Omron CX-Programmer project NewProject (CX-Programmer 9.75)

# PLC NewPLC1: CP2E-N N

## Global symbols (name address type ; comment)
ABNRML_INDICATOR 101.06 BOOL  ; ABNORMAL_IND
AIR_PRESS_OK 0.01 BOOL  ; AIR_PRESS_OK
AUTO_SS 1.09 BOOL  ; AUTO SS
1.08 BOOL  ; manual_press
4 CHANNEL  ; LVDT1_INP_POS
5 CHANNEL  ; LVDT2_INP_POS
D100 CHANNEL  ; LVDT1_CURRENT_VAL_MM
D1000 CHANNEL  ; lvdt1_max_hmi_log
D1002 CHANNEL  ; lvdt1_min_hmi_log
D1004 CHANNEL  ; lvdt2_max_hmi_log
D1006 CHANNEL  ; lvdt2_min_hmi_log
D1010 CHANNEL  ; lvdt1_max_hmi_log.
D1012 CHANNEL  ; lvdt1_min_hmi_log.
D1014 CHANNEL  ; lvdt2_max_hmi_log.
D1016 CHANNEL  ; lvdt2_min_hmi_log.
D110 CHANNEL  ; LVDT2_CURRENT_VAL_MM
D1230 CHANNEL  ; servo_pulse.
D1240 CHANNEL  ; LVDT1_CURRENT_VAL_MM.
D1250 CHANNEL  ; LVDT2_CURRENT_VAL_MM.
D1280 CHANNEL  ; LVDT_POS_OK_PART
D1300 CHANNEL  ; rpm_hmi
D1305 CHANNEL  ; .
D1310 CHANNEL  ; servo_freq.
D150 CHANNEL  ; TOTAL PULSES FOR ROTATION
D1520 CHANNEL  ; PART2_CAL
D1550 CHANNEL  ; PART2_CAL.
D1700 CHANNEL  ; SERVO_PV
D20 CHANNEL  ; CYCLE TIME
D200 CHANNEL  ; UPPER_LIMIT_M1_HMI
D2000 CHANNEL  ; TOTAL_NG_GEAR_RUNOUT_LOWER_LIM
D2002 CHANNEL  ; TOTAL_NG_GEAR_RUNOUT_UPPER_LIM
D202 CHANNEL  ; LOWER_LIMIT_1_HMI
D204 CHANNEL  ; UPPER_LIMIT_M2_HMI
D206 CHANNEL  ; LOWER_LIMIT_M2_HMI
D210 CHANNEL  ; OFFSET_M1_HMI
D212 CHANNEL  ; OFFSET._M1_HMI
D214 CHANNEL  ; OFFSET_M2_HMI
D216 CHANNEL  ; OFFSET._M2_HMI
D22 CHANNEL  ; OK_COUNT
D220 CHANNEL  ; FINAL_UPPER_LIMIT
D222 CHANNEL  ; FINAL_LOWER_LIMIT
D224 CHANNEL  ; FINAL_LOWER_LIMIT
D230 CHANNEL  ; LOWER_LIMIT_1_HMI
D240 CHANNEL  ; LOWER_LIMIT_1_HMI
D25 CHANNEL  ; NG_COUNT
D250 CHANNEL  ; UPPER_LIMIT_M2_HMI
D260 CHANNEL  ; OFFSET_M2_HMI
D270 CHANNEL  ; LOWER_LIMIT_M2_HMI
D280 CHANNEL  ; OFFSET._M2_HMI
D300 CHANNEL  ; WORD LAMP STATUS
D550 CHANNEL  ; LVDT1_INP_POS.
D555 CHANNEL  ; LVDT2_INP_POS.
D570 CHANNEL  ; OFFSET_LVDT
D575 CHANNEL  ; LVDT2_CUR_VAL
D590 CHANNEL  ; OFFSET
D595 CHANNEL  ; LVDT1_CUR_VAL
D605 CHANNEL  ; .
D7055 CHANNEL  ; LVDT1_MAX_HMI
D820 CHANNEL  ; rot_degree
D830 CHANNEL  ; PART1_SERVOCOUNT_HMI
D840 CHANNEL  ; PART2_SERVOCOUNT_HMI
D850 CHANNEL  ; rot_deg.
D900 CHANNEL  ; LVDT2_MAX_HMI
D902 CHANNEL  ; LVDT1_MAX_HMI
D904 CHANNEL  ; LVDT2_MIN_HMI
D906 CHANNEL  ; LVDT1_Min_HMI
D910 CHANNEL  ; LVDT2_MAX_HMI
D910 CHANNEL  ; LVDT1_MAX_HMI
D920 CHANNEL  ; servo_float
D930 CHANNEL  ; part1_fullbody_servocount
D930 CHANNEL  ; PART1_FULLBODY_PULSE
D940 CHANNEL  ; PART2_FULLBODY_SERVOCOUNT
D950 CHANNEL  ; LVDT1_Min_HMI
T046 BOOL  ; delay time for lvdt to adjust
W10.00 BOOL  ; CYCLE START
W11.00 BOOL  ; PART_FEEDER_UP_BIT
W11.01 BOOL  ; PART_HOLDER_FWD_BIT
W11.02 BOOL  ; PART_FEED_DONE_FLAG
W11.03 BOOL  ; TEST_CYCLE_START
W11.04 BOOL  ; LVDT_TEST_POSITION
W11.05 BOOL  ; SERVO_CMD1
W11.06 BOOL  ; TEST_DONE_FLAG_OK
W11.07 BOOL  ; CYCLE_COMPLETING_OK_process_start
W11.08 BOOL  ; PART_FEEDER_UP_OK
W11.09 BOOL  ; CYCLE_COM_OK_flag
W11.10 BOOL  ; LVDT_PUSHER_FWD_OK
W12.00 BOOL  ; TYPENO._1
W12.01 BOOL  ; TYPNO._2
W12.02 BOOL  ; PART1
W12.03 BOOL  ; PART2
W13.06 BOOL  ; TEST_DONE_FLAG_NG
W13.07 BOOL  ; CYCLE_COMPLETING_NG_process_start
W13.08 BOOL  ; PART_FEEDER_UP_NG
W13.09 BOOL  ; CYCLE_COM_NG
W13.10 BOOL  ; LVDT_PUSHER_fwd_NG
W14.00 BOOL  ; BIO_SCAN_OK
W15.00 BOOL  ; NG_FLAG
W15.01 BOOL  ; OK_FLAG
W16.00 BOOL  ; PART_FEEDER_DN_BIT
W16.01 BOOL  ; PART_HOLDER_REV_BIT
W16.04 BOOL  ; LVDT_CYL_REV_ok
W16.08 BOOL  ; PART_FEED_DN_BIT_OK
W16.10 BOOL  ; LVDT_PUSHER_REV_BIT
W17.01 BOOL  ; PART_HOLDER_REV__NG_BIT
W17.04 BOOL  ; LVDT_CYL_REV_NG
W17.08 BOOL  ; PART_FEEDER_DN_NG
W17.10 BOOL  ; LVDT_PUSHER_REV_NG
W18.04 BOOL  ; LVDT_CYL_REV_EMG
W19.00 BOOL  ; BUZZER_NG_PART
W19.01 BOOL  ; BUZZER_BIT
W19.03 BOOL  ; ng_bin_sensor
W22.00 BOOL  ; PART_FEED_UP_MAN
W22.01 BOOL  ; PART_FEED_DN_MAN
W22.02 BOOL  ; PART_HOLD1_FWD_MAN
W22.03 BOOL  ; PART_HOLD2_FWD_MAN
W22.04 BOOL  ; PART_HOLD1_REV_MAN
W22.05 BOOL  ; PART_HOLD2_REV_MAN
W22.06 BOOL  ; LVDT_FWD_MAN
W22.07 BOOL  ; LVDT_REV_MAN
W22.08 BOOL  ; LVDT_PUSH_FWD_MAN
W22.09 BOOL  ; LVDT_PUSH_REV_MAN
W23.00 BOOL  ; PART_FEED_UP_MAN
W23.01 BOOL  ; PART_FEED_DN_MAN
W23.02 BOOL  ; PART_HOLD1_FWD_MAN
W23.03 BOOL  ; PART_HOLD2_FWD_MAN
W23.04 BOOL  ; PART_HOLD1_REV_MAN
W23.05 BOOL  ; PART_HOLD2_REV_MAN
W23.06 BOOL  ; LVDT_FWD_MAN
W23.07 BOOL  ; LVDT_REV_MAN
W23.08 BOOL  ; LVDT_PUSH_FWD_MAN
W23.09 BOOL  ; LVDT_PUSH_REV_MAN
W24.00 BOOL  ; FULL_PART_TESTED
W25.00 BOOL  ; LVDT_ORIGIN
W25.01 BOOL  ; PART_HOLDER_ORIGIN
W25.02 BOOL  ; PART_FEEDER_ORIGIN
W25.03 BOOL  ; LVDT_PUSHER_FWD
W25.04 BOOL  ; LVDT_PUSHER_HM
W25.12 BOOL  ; part_feeder_up_org
W25.15 BOOL  ; PUSHER_HOME_ORG
W26.00 BOOL  ; MASTER_ON_BIT
W26.01 BOOL  ; SERVO_MAN
W26.02 BOOL  ; LVDT_HOME
W26.12 BOOL  ; servo_man
W2.06 BOOL  ; BIO_SCANNED
W2.08 BOOL  ; RESET_ORG
W30.00 BOOL  ; COUNTER_RESET_HMI
W32.00 BOOL  ; servo_cmd2
W39.01 BOOL  ; WRONG MODEL SELECTED
W50.00 BOOL  ; PART_FEEDER_UP_RS_ABS/ CYL NOT UP
W50.01 BOOL  ; PART_FEEDER_DN_RS_ABS/CYL NOT DN
W50.02 BOOL  ; PART_HOLD_CLOSE_RS_ABS/ PART NOT HOLD
W50.03 BOOL  ; PART_HOLD_OPEN_RS_ABS/ PART NOT RELEASED
W50.04 BOOL  ; LVDT1_TEST_RS_ABS/ LVDT1 NOT AT TEST POS
W50.05 BOOL  ; LVDT2_TEST_RS_ABS/ LVDT2 NOT AT TEST POS
W50.06 BOOL  ; LVDT1_HM_RS_ABS/ LVDT1 NOT AT HOME POS
W50.07 BOOL  ; LVDT2_HM_RS_ABS/ LVDT2 NOT AT HOME POS
W50.08 BOOL  ; PUSHER LIM RS ABS / PUSHER NOT MOVING FWD
W50.09 BOOL  ; PUSHER HOME RS ABSENT / PUSHER NOT MOVING REV
W50.10 BOOL  ; CHECK_PART_CLAMP_RS/PART SELECTION RS ERROR
W55.00 BOOL  ; servo_run1_complete_flag
W55.01 BOOL  ; lvdt_ready_for_test
W55.02 BOOL  ; NGpart_ready_to_remove
W55.03 BOOL  ; OKpart_ready_to_remove
W55.04 BOOL  ; LVDT_PUSHING_DONE
W55.05 BOOL  ; PAR_UNCLAMP_DONE_OK
W55.06 BOOL  ; LVDT_PUSH_DONE_NG
W55.07 BOOL  ; PAR_UNCLAMP_DONE_NG
W55.08 BOOL  ; NGpart_ready_to_remove
W55.10 BOOL  ; lvdt_home
W56.01 BOOL  ; servo_ready_for_cmd2
W60.10 BOOL  ; PART_NOT_MATCHED
W60.11 BOOL  ; PART1_MATCHED
W60.12 BOOL  ; PART_2_MATCHED
W6.00 BOOL  ; LOG_PART1_RESULT
W6.01 BOOL  ; LOG_PART2_RESULT
W70.00 BOOL  ; EMG_ALARM
W70.01 BOOL  ; AIR_PRESS_ALARM
W70.02 BOOL  ; SAFETY_DOOR_ALARM
W70.03 BOOL  ; PART_ABSENT_ALARM
W70.04 BOOL  ; PART_NOT_MATCH_ALARM
W76.01 BOOL  ; part2_match
W77.01 BOOL  ; not_match
W78.01 BOOL  ; not_match.
W79.01 BOOL  ; part1_match
W80.00 BOOL  ; ABNORMAL_LIGHT
W80.03 BOOL  ; PART_NOT_PRESENT_ALARM
W80.04 BOOL  ; NG_PART_ALARM
W8.00 BOOL  ; LVDT_PUSHED_flag
W8.01 BOOL  ; LVDT_PUSH_DONE
W9.00 BOOL  ; MACHINE_HOME
W9.01 BOOL  ; LVDT_PUSH_ONCE
W9.02 BOOL  ; LVDT_PUSH_RTN
W9.03 BOOL  ; LVDT_PUSHED_FLAG
W9.04 BOOL  ; CYCLE READY_FLAG
W9.05 BOOL  ; servo_cmd3
W9.06 BOOL  ; part_ok_HMI
W9.07 BOOL  ; part_ng_HMI
BIO_SCAN 0.00 BOOL  ; BIOMETRIC
DUAL_PB1 1.11 BOOL  ; DUAL_PB1
DUAL_PB2 2.00 BOOL  ; DUAL_PB2
EMG_LAMP 101.03 BOOL  ; EMG_LAMP
EMG_PB 2.04 BOOL  ; EMG_PB
LVDT1_HOME_RS 0.05 BOOL  ; LVDT1_HM_RS
LVDT1_TEST_RS 0.04 BOOL  ; LVDT1_TST_RS
LVDT2_HOME_RS 0.07 BOOL  ; LVDT2_HM_RS
LVDT2_TEST_RS 0.06 BOOL  ; LVDT2_TST_RS
LVDT_CYL_FWD 100.06 BOOL  ; LVDT_CYL_FWD
LVDT_CYL_REV 100.07 BOOL  ; LVDT_CYL_REV
LVDT_PUSHER_FWD 101.00 BOOL  ; LVDT_PUSH_CYL_FWD
LVDT_PUSHER_REV 101.01 BOOL  ; LVDT_PUSH_CYL_REV
LVDT_PUSH_HOME 2.06 BOOL  ; LVDT_PUSH_HOME
LVDT_PUSH_LIM 2.05 BOOL  ; LVDT_PUSHER_LIM
MANUAL_SS 1.10 BOOL  ; MANUAL_SS
MASTER_LAMP 101.04 BOOL  ; MASTER_LAMP
MODEL_2 1.02 BOOL  ; 2
NG_BIN_SEN 0.11 BOOL  ; NG_BIN_SENSOR
NG_BUZZER 101.02 BOOL  ; NG_BUZZER
NG_UNCLAMP_PB 2.02 BOOL  ; NG_UNCLAMP_PB
ORGN_INDICATOR 101.05 BOOL  ; ORIGIN_IND
ORIGIN_RETURN_PB 2.01 BOOL  ; ORIGIN_RETURN_PB
PART_1 1.00 BOOL  ; PART_1
PART_2 1.01 BOOL  ; PART_2
PART_CLAMP_CLOSE_P2 2.10 BOOL  ; PART_CLAMP_CLOSE_P2
PART_FEEDER_DN 103.01 BOOL  ; PART_FEEDER_DOWN
PART_FEEDER_UP 103.00 BOOL  ; PART_FEEDER_UP
PART_FEED_DN_RS 2.08 BOOL  ; PART_FEEDER_DN_RS
PART_FEED_UP_RS 2.07 BOOL  ; PART_FEEDER_UP_RS
PART_HOLD1_CLOSE_RS 0.02 BOOL  ; PART_HOLDER_FRONT_RS
PART_HOLD1_OPEN_RS 0.03 BOOL  ; PART_HOLDER_BACK_RS
PART_HOLD2_CLOSE_RS 0.08 BOOL  ; part_holde2_close_rs
PART_HOLD2_OPEN_RS 0.09 BOOL  ; part_holder2_open_rs
PART_HOLDER1_FWD 100.01 BOOL  ; PART_HOLDER1_FWD
PART_HOLDER1_REV 100.03 BOOL  ; PART_HOLDER1_REV
PART_HOLDER2_FWD 100.04 BOOL  ; PART_HOLDER2_FWD
PART_HOLDER2_REV 100.05 BOOL  ; PART_HOLDER2_REV
PART_PRESENCE_SENSOR 2.11 BOOL  ; PART_PRESENCE_SENSOR
RESET_PB 2.03 BOOL  ; RESET_PB
SAFETY_LIM1 2.09 BOOL  ; SAFETY_LIM1
SERVO_DIR 100.01 BOOL  ; SERVO_DIRECTION
SERVO_OUT 102.04 BOOL  ; SERVO
SERVO_PULSE 100.00 BOOL  ; SERVO_PULSE
TEST_READY_SENSOR 3.00 BOOL  ; PART_READY FOR TEST SENSOR
TOWER_LIGHT 101.07 BOOL  ; TOWER_LIGHT
master_start 0.10 BOOL  ; START_PB

## Program NewProgram1 (cyclic task 0)
Local symbols
ILC BOOL
MODEL_3 BOOL
PART_UNHOLD BOOL
cf11e BOOL
dsc BOOL

### Section IN_OUT

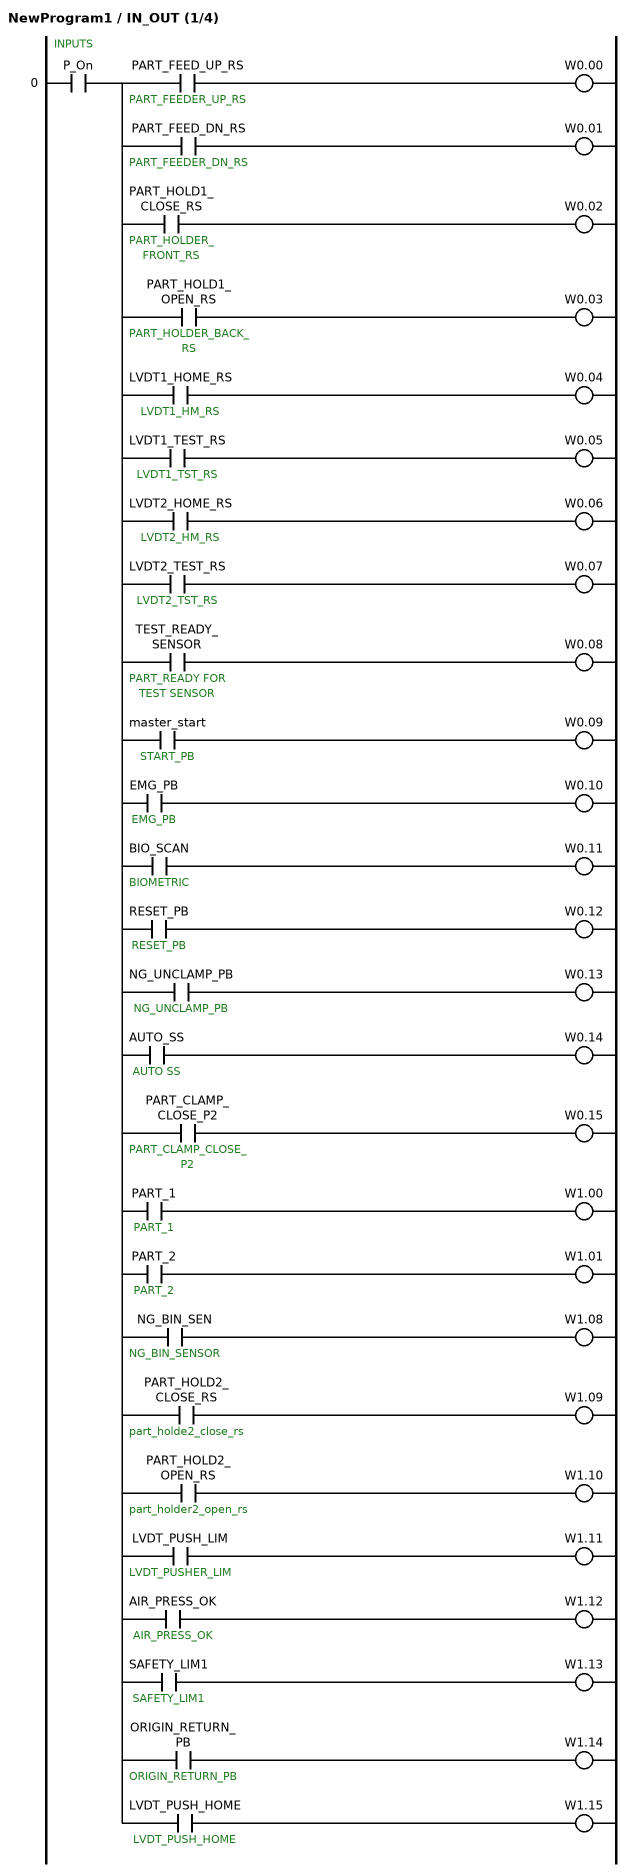
; rung 0: INPUTS
LD P_On
OUT TR0
AND PART_FEED_UP_RS  ; PART_FEEDER_UP_RS
OUT W0.00
LD TR0
AND PART_FEED_DN_RS  ; PART_FEEDER_DN_RS
OUT W0.01
LD TR0
AND PART_HOLD1_CLOSE_RS  ; PART_HOLDER_FRONT_RS
OUT W0.02
LD TR0
AND PART_HOLD1_OPEN_RS  ; PART_HOLDER_BACK_RS
OUT W0.03
LD TR0
AND LVDT1_HOME_RS  ; LVDT1_HM_RS
OUT W0.04
LD TR0
AND LVDT1_TEST_RS  ; LVDT1_TST_RS
OUT W0.05
LD TR0
AND LVDT2_HOME_RS  ; LVDT2_HM_RS
OUT W0.06
LD TR0
AND LVDT2_TEST_RS  ; LVDT2_TST_RS
OUT W0.07
LD TR0
AND TEST_READY_SENSOR  ; PART_READY FOR TEST SENSOR
OUT W0.08
LD TR0
AND master_start  ; START_PB
OUT W0.09
LD TR0
AND EMG_PB  ; EMG_PB
OUT W0.10
LD TR0
AND BIO_SCAN  ; BIOMETRIC
OUT W0.11
LD TR0
AND RESET_PB  ; RESET_PB
OUT W0.12
LD TR0
AND NG_UNCLAMP_PB  ; NG_UNCLAMP_PB
OUT W0.13
LD TR0
AND AUTO_SS  ; AUTO SS
OUT W0.14
LD TR0
AND PART_CLAMP_CLOSE_P2  ; PART_CLAMP_CLOSE_P2
OUT W0.15
LD TR0
AND PART_1  ; PART_1
OUT W1.00
LD TR0
AND PART_2  ; PART_2
OUT W1.01
LD TR0
AND NG_BIN_SEN  ; NG_BIN_SENSOR
OUT W1.08
LD TR0
AND PART_HOLD2_CLOSE_RS  ; part_holde2_close_rs
OUT W1.09
LD TR0
AND PART_HOLD2_OPEN_RS  ; part_holder2_open_rs
OUT W1.10
LD TR0
AND LVDT_PUSH_LIM  ; LVDT_PUSHER_LIM
OUT W1.11
LD TR0
AND AIR_PRESS_OK  ; AIR_PRESS_OK
OUT W1.12
LD TR0
AND SAFETY_LIM1  ; SAFETY_LIM1
OUT W1.13
LD TR0
AND ORIGIN_RETURN_PB  ; ORIGIN_RETURN_PB
OUT W1.14
LD TR0
AND LVDT_PUSH_HOME  ; LVDT_PUSH_HOME
OUT W1.15

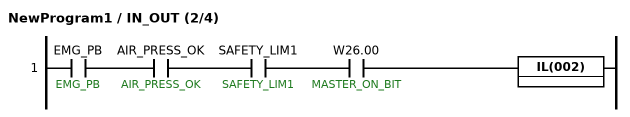
; rung 1
LD EMG_PB  ; EMG_PB
AND AIR_PRESS_OK  ; AIR_PRESS_OK
AND SAFETY_LIM1  ; SAFETY_LIM1
AND W26.00  ; MASTER_ON_BIT
IL(002)

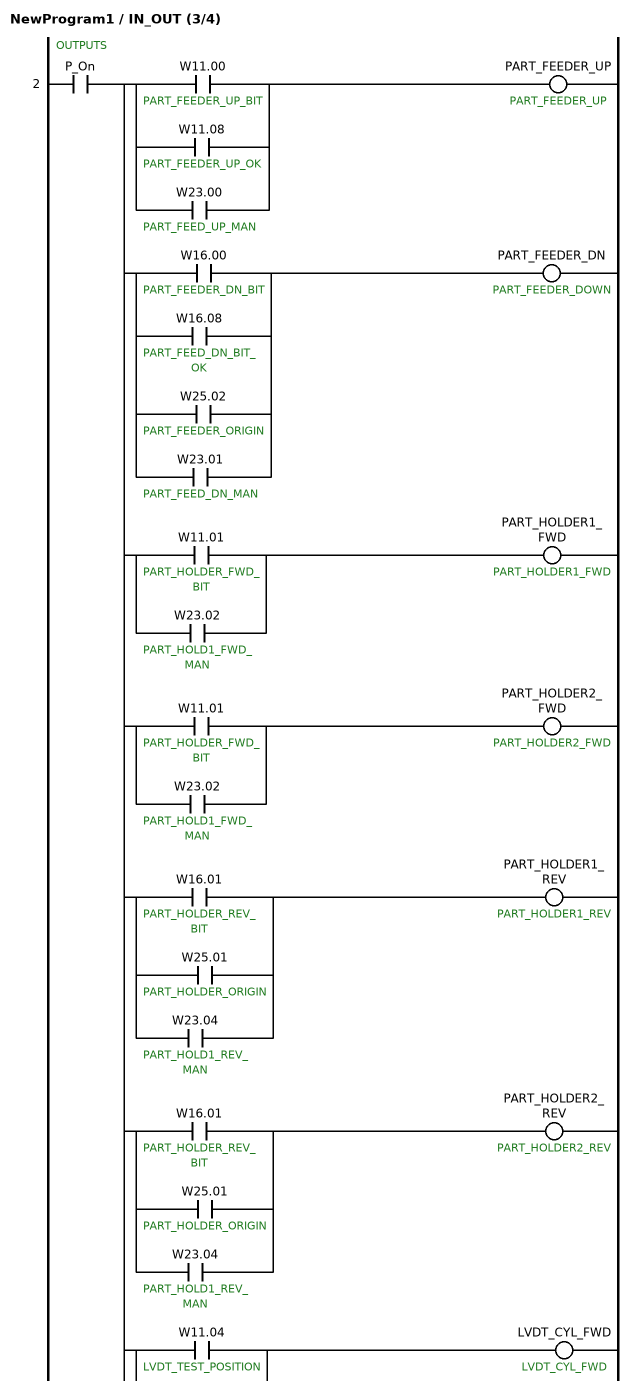

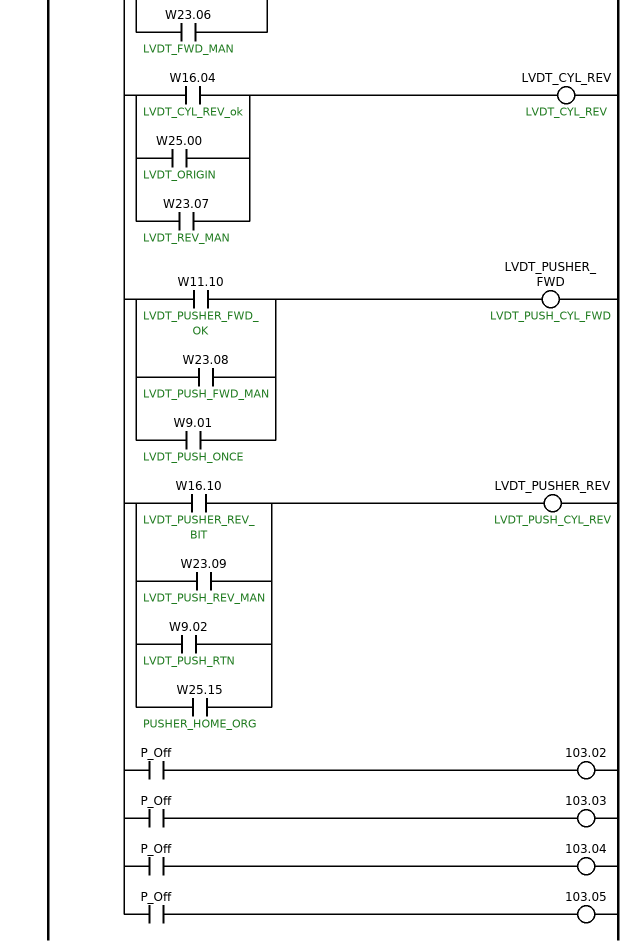
; rung 2: OUTPUTS
LD P_On
OUT TR0
LD W11.00  ; PART_FEEDER_UP_BIT
OR W11.08  ; PART_FEEDER_UP_OK
OR W23.00  ; PART_FEED_UP_MAN
ANDLD
OUT PART_FEEDER_UP  ; PART_FEEDER_UP
LD TR0
LD W16.00  ; PART_FEEDER_DN_BIT
OR W16.08  ; PART_FEED_DN_BIT_OK
OR W25.02  ; PART_FEEDER_ORIGIN
OR W23.01  ; PART_FEED_DN_MAN
ANDLD
OUT PART_FEEDER_DN  ; PART_FEEDER_DOWN
LD TR0
LD W11.01  ; PART_HOLDER_FWD_BIT
OR W23.02  ; PART_HOLD1_FWD_MAN
ANDLD
OUT PART_HOLDER1_FWD  ; PART_HOLDER1_FWD
LD TR0
LD W11.01  ; PART_HOLDER_FWD_BIT
OR W23.02  ; PART_HOLD1_FWD_MAN
ANDLD
OUT PART_HOLDER2_FWD  ; PART_HOLDER2_FWD
LD TR0
LD W16.01  ; PART_HOLDER_REV_BIT
OR W25.01  ; PART_HOLDER_ORIGIN
OR W23.04  ; PART_HOLD1_REV_MAN
ANDLD
OUT PART_HOLDER1_REV  ; PART_HOLDER1_REV
LD TR0
LD W16.01  ; PART_HOLDER_REV_BIT
OR W25.01  ; PART_HOLDER_ORIGIN
OR W23.04  ; PART_HOLD1_REV_MAN
ANDLD
OUT PART_HOLDER2_REV  ; PART_HOLDER2_REV
LD TR0
LD W11.04  ; LVDT_TEST_POSITION
OR W23.06  ; LVDT_FWD_MAN
ANDLD
OUT LVDT_CYL_FWD  ; LVDT_CYL_FWD
LD TR0
LD W16.04  ; LVDT_CYL_REV_ok
OR W25.00  ; LVDT_ORIGIN
OR W23.07  ; LVDT_REV_MAN
ANDLD
OUT LVDT_CYL_REV  ; LVDT_CYL_REV
LD TR0
LD W11.10  ; LVDT_PUSHER_FWD_OK
OR W23.08  ; LVDT_PUSH_FWD_MAN
OR W9.01  ; LVDT_PUSH_ONCE
ANDLD
OUT LVDT_PUSHER_FWD  ; LVDT_PUSH_CYL_FWD
LD TR0
LD W16.10  ; LVDT_PUSHER_REV_BIT
OR W23.09  ; LVDT_PUSH_REV_MAN
OR W9.02  ; LVDT_PUSH_RTN
OR W25.15  ; PUSHER_HOME_ORG
ANDLD
OUT LVDT_PUSHER_REV  ; LVDT_PUSH_CYL_REV
LD TR0
AND P_Off
OUT 103.02
LD TR0
AND P_Off
OUT 103.03
LD TR0
AND P_Off
OUT 103.04
LD TR0
AND P_Off
OUT 103.05

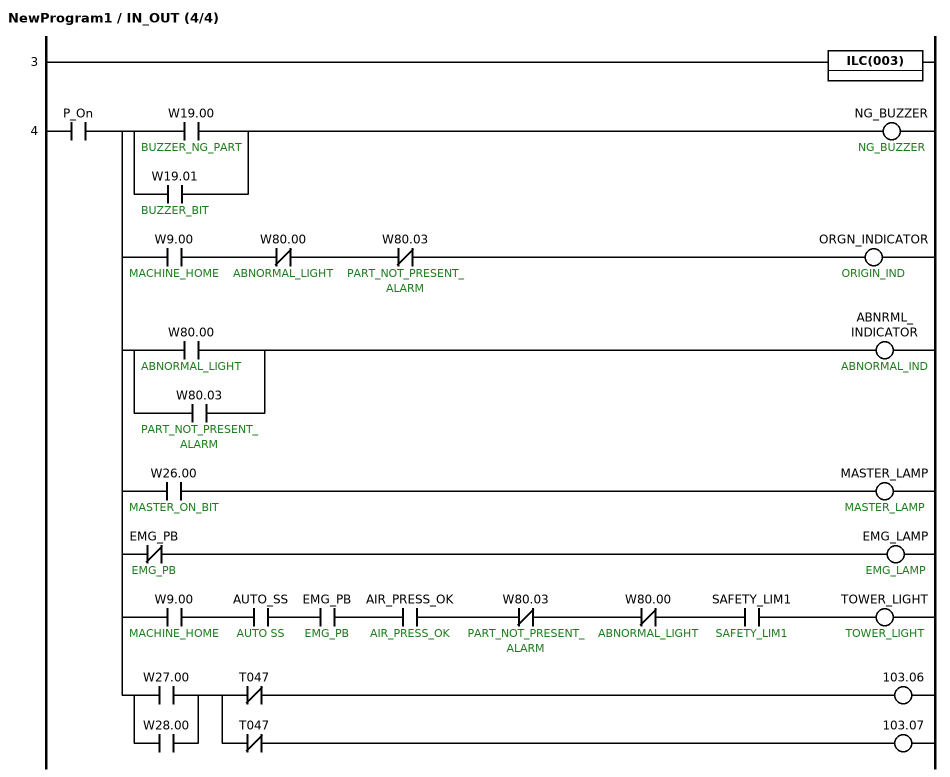
; rung 3
ILC(003)
; rung 4
LD P_On
OUT TR0
LD W19.00  ; BUZZER_NG_PART
OR W19.01  ; BUZZER_BIT
ANDLD
OUT NG_BUZZER  ; NG_BUZZER
LD TR0
AND W9.00  ; MACHINE_HOME
ANDNOT W80.00  ; ABNORMAL_LIGHT
ANDNOT W80.03  ; PART_NOT_PRESENT_ALARM
OUT ORGN_INDICATOR  ; ORIGIN_IND
LD TR0
LD W80.00  ; ABNORMAL_LIGHT
OR W80.03  ; PART_NOT_PRESENT_ALARM
ANDLD
OUT ABNRML_INDICATOR  ; ABNORMAL_IND
LD TR0
AND W26.00  ; MASTER_ON_BIT
OUT MASTER_LAMP  ; MASTER_LAMP
LD TR0
ANDNOT EMG_PB  ; EMG_PB
OUT EMG_LAMP  ; EMG_LAMP
LD TR0
AND W9.00  ; MACHINE_HOME
AND AUTO_SS  ; AUTO SS
AND EMG_PB  ; EMG_PB
AND AIR_PRESS_OK  ; AIR_PRESS_OK
ANDNOT W80.03  ; PART_NOT_PRESENT_ALARM
ANDNOT W80.00  ; ABNORMAL_LIGHT
AND SAFETY_LIM1  ; SAFETY_LIM1
OUT TOWER_LIGHT  ; TOWER_LIGHT
LD TR0
LD W27.00
OR W28.00
ANDLD
OUT TR0
ANDNOT T047
OUT 103.06
LD TR0
ANDNOT T047
OUT 103.07

### Section AUTO

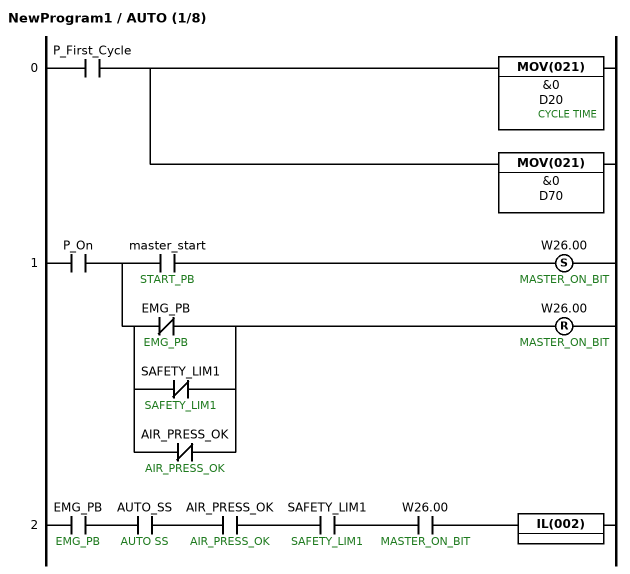
; rung 0
LD P_First_Cycle
MOV(021) &0 D20  ; CYCLE TIME
MOV(021) &0 D70
; rung 1
LD P_On
OUT TR0
AND master_start  ; START_PB
SET W26.00  ; MASTER_ON_BIT
LD TR0
LDNOT EMG_PB  ; EMG_PB
ORNOT SAFETY_LIM1  ; SAFETY_LIM1
ORNOT AIR_PRESS_OK  ; AIR_PRESS_OK
ANDLD
RSET W26.00  ; MASTER_ON_BIT
; rung 2
LD EMG_PB  ; EMG_PB
AND AUTO_SS  ; AUTO SS
AND AIR_PRESS_OK  ; AIR_PRESS_OK
AND SAFETY_LIM1  ; SAFETY_LIM1
AND W26.00  ; MASTER_ON_BIT
IL(002)

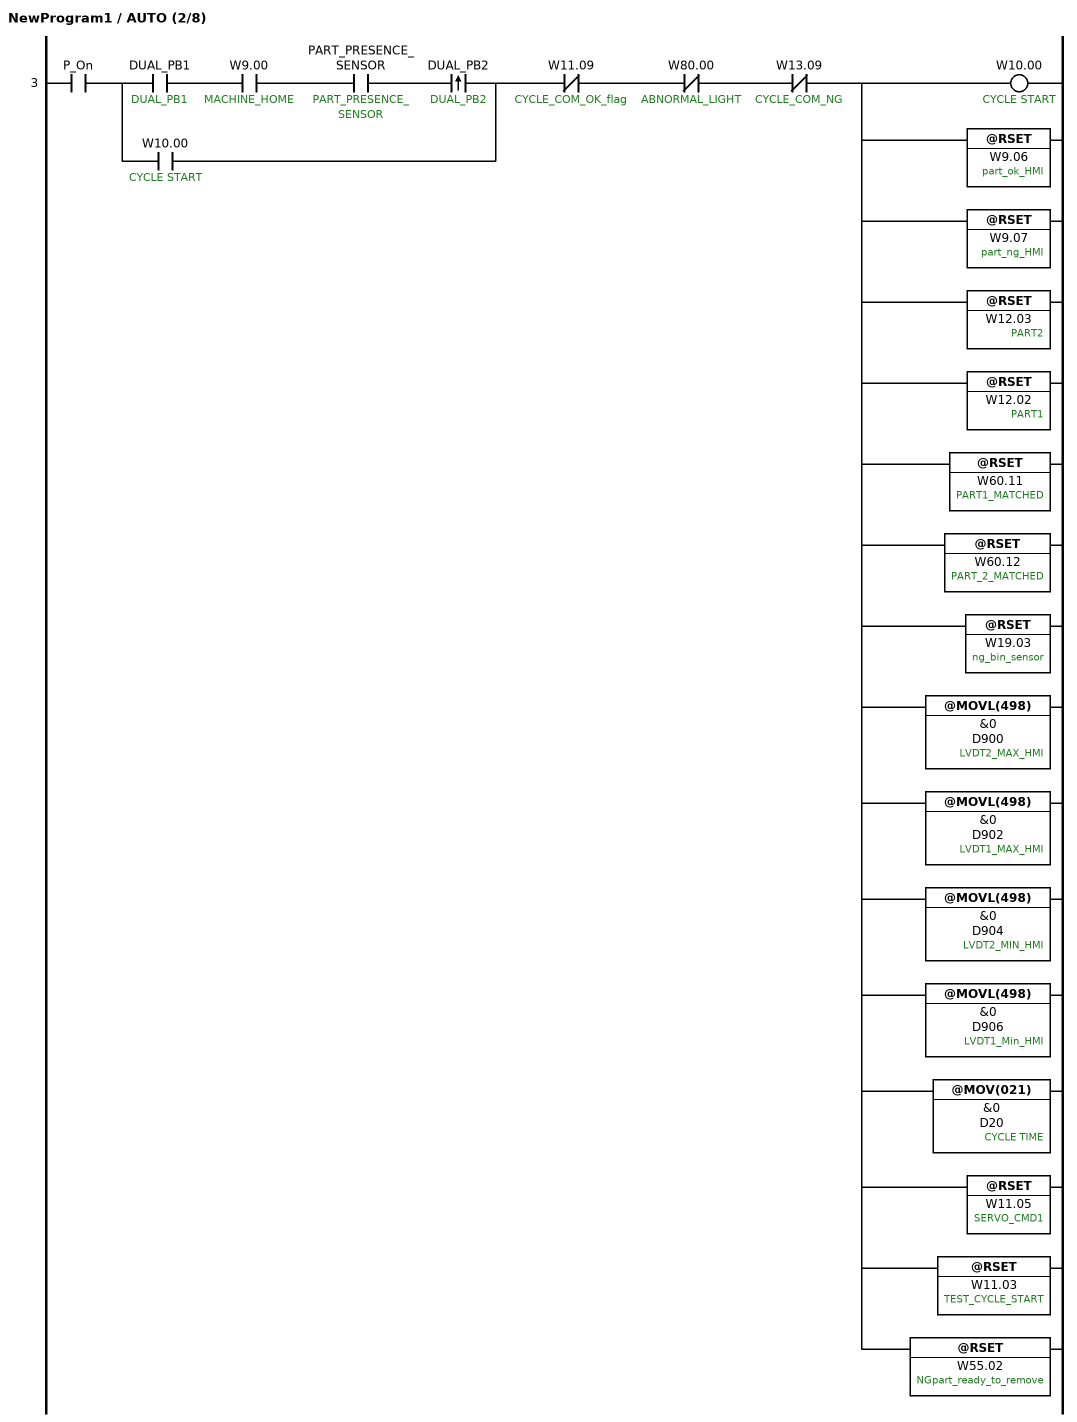
; rung 3
LD P_On
LD DUAL_PB1  ; DUAL_PB1
AND W9.00  ; MACHINE_HOME
AND PART_PRESENCE_SENSOR  ; PART_PRESENCE_SENSOR
@AND DUAL_PB2  ; DUAL_PB2
OR W10.00  ; CYCLE START
ANDLD
ANDNOT W11.09  ; CYCLE_COM_OK_flag
ANDNOT W80.00  ; ABNORMAL_LIGHT
ANDNOT W13.09  ; CYCLE_COM_NG
OUT W10.00  ; CYCLE START
@RSET W9.06  ; part_ok_HMI
@RSET W9.07  ; part_ng_HMI
@RSET W12.03  ; PART2
@RSET W12.02  ; PART1
@RSET W60.11  ; PART1_MATCHED
@RSET W60.12  ; PART_2_MATCHED
@RSET W19.03  ; ng_bin_sensor
@MOVL(498) &0 D900  ; LVDT2_MAX_HMI
@MOVL(498) &0 D902  ; LVDT1_MAX_HMI
@MOVL(498) &0 D904  ; LVDT2_MIN_HMI
@MOVL(498) &0 D906  ; LVDT1_Min_HMI
@MOV(021) &0 D20  ; CYCLE TIME
@RSET W11.05  ; SERVO_CMD1
@RSET W11.03  ; TEST_CYCLE_START
@RSET W55.02  ; NGpart_ready_to_remove

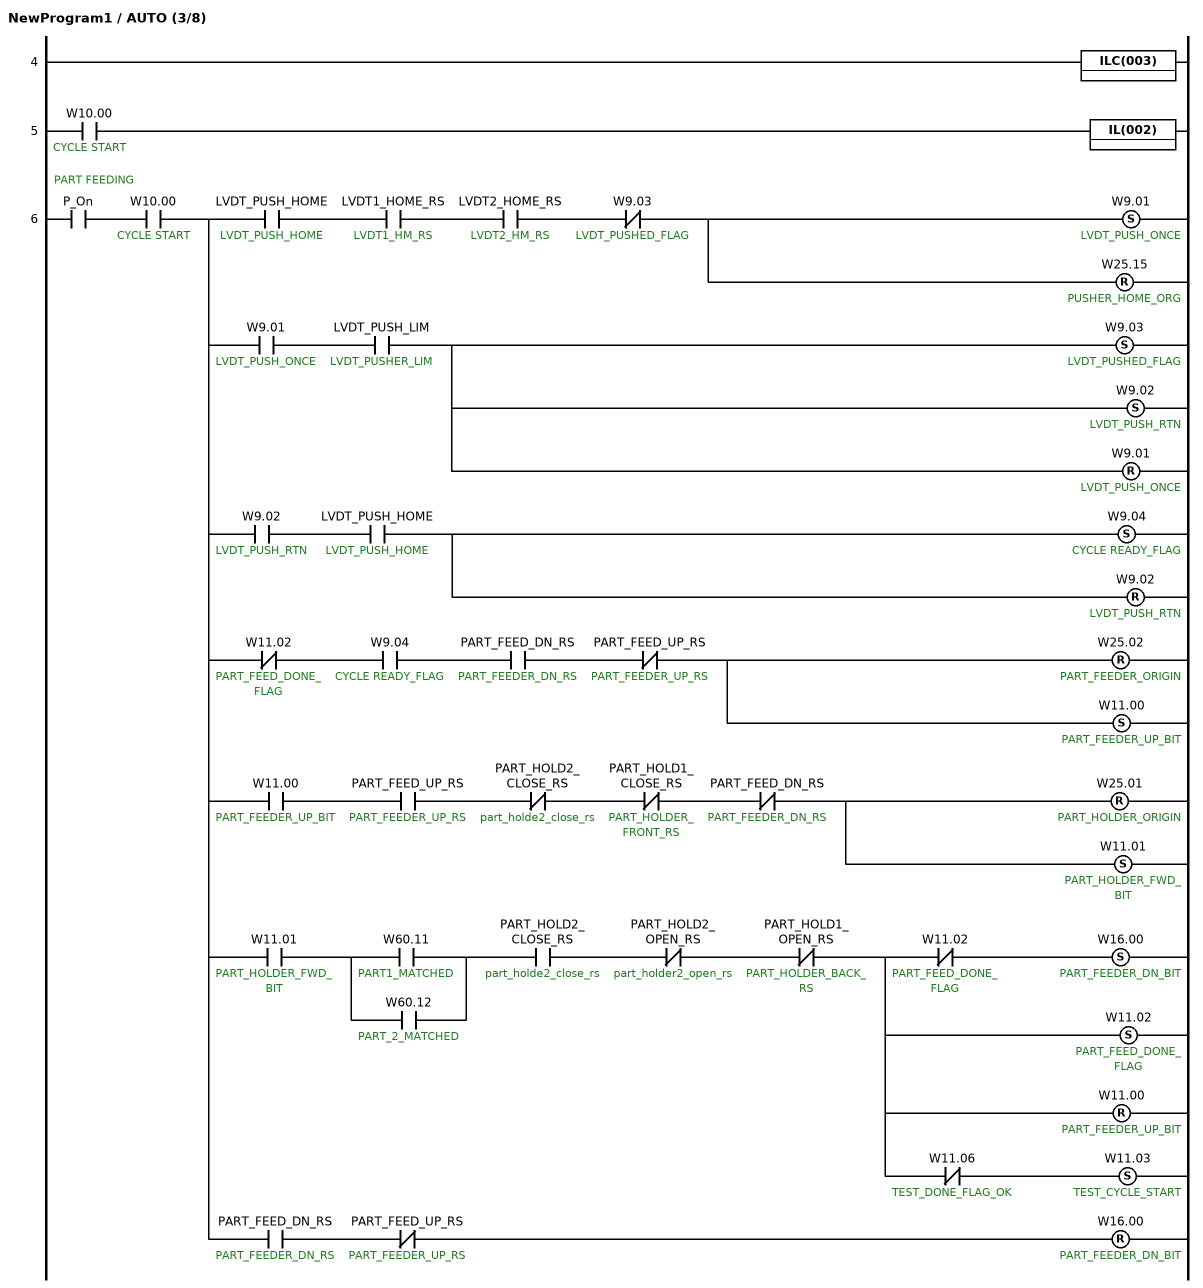
; rung 4
ILC(003)
; rung 5
LD W10.00  ; CYCLE START
IL(002)
; rung 6: PART FEEDING
LD P_On
AND W10.00  ; CYCLE START
OUT TR0
AND LVDT_PUSH_HOME  ; LVDT_PUSH_HOME
AND LVDT1_HOME_RS  ; LVDT1_HM_RS
AND LVDT2_HOME_RS  ; LVDT2_HM_RS
ANDNOT W9.03  ; LVDT_PUSHED_FLAG
SET W9.01  ; LVDT_PUSH_ONCE
RSET W25.15  ; PUSHER_HOME_ORG
LD TR0
AND W9.01  ; LVDT_PUSH_ONCE
AND LVDT_PUSH_LIM  ; LVDT_PUSHER_LIM
SET W9.03  ; LVDT_PUSHED_FLAG
SET W9.02  ; LVDT_PUSH_RTN
RSET W9.01  ; LVDT_PUSH_ONCE
LD TR0
AND W9.02  ; LVDT_PUSH_RTN
AND LVDT_PUSH_HOME  ; LVDT_PUSH_HOME
SET W9.04  ; CYCLE READY_FLAG
RSET W9.02  ; LVDT_PUSH_RTN
LD TR0
ANDNOT W11.02  ; PART_FEED_DONE_FLAG
AND W9.04  ; CYCLE READY_FLAG
AND PART_FEED_DN_RS  ; PART_FEEDER_DN_RS
ANDNOT PART_FEED_UP_RS  ; PART_FEEDER_UP_RS
RSET W25.02  ; PART_FEEDER_ORIGIN
SET W11.00  ; PART_FEEDER_UP_BIT
LD TR0
AND W11.00  ; PART_FEEDER_UP_BIT
AND PART_FEED_UP_RS  ; PART_FEEDER_UP_RS
ANDNOT PART_HOLD2_CLOSE_RS  ; part_holde2_close_rs
ANDNOT PART_HOLD1_CLOSE_RS  ; PART_HOLDER_FRONT_RS
ANDNOT PART_FEED_DN_RS  ; PART_FEEDER_DN_RS
RSET W25.01  ; PART_HOLDER_ORIGIN
SET W11.01  ; PART_HOLDER_FWD_BIT
LD TR0
AND W11.01  ; PART_HOLDER_FWD_BIT
LD W60.11  ; PART1_MATCHED
OR W60.12  ; PART_2_MATCHED
ANDLD
AND PART_HOLD2_CLOSE_RS  ; part_holde2_close_rs
ANDNOT PART_HOLD2_OPEN_RS  ; part_holder2_open_rs
ANDNOT PART_HOLD1_OPEN_RS  ; PART_HOLDER_BACK_RS
OUT TR1
ANDNOT W11.02  ; PART_FEED_DONE_FLAG
SET W16.00  ; PART_FEEDER_DN_BIT
LD TR1
SET W11.02  ; PART_FEED_DONE_FLAG
RSET W11.00  ; PART_FEEDER_UP_BIT
ANDNOT W11.06  ; TEST_DONE_FLAG_OK
SET W11.03  ; TEST_CYCLE_START
LD TR0
AND PART_FEED_DN_RS  ; PART_FEEDER_DN_RS
ANDNOT PART_FEED_UP_RS  ; PART_FEEDER_UP_RS
RSET W16.00  ; PART_FEEDER_DN_BIT

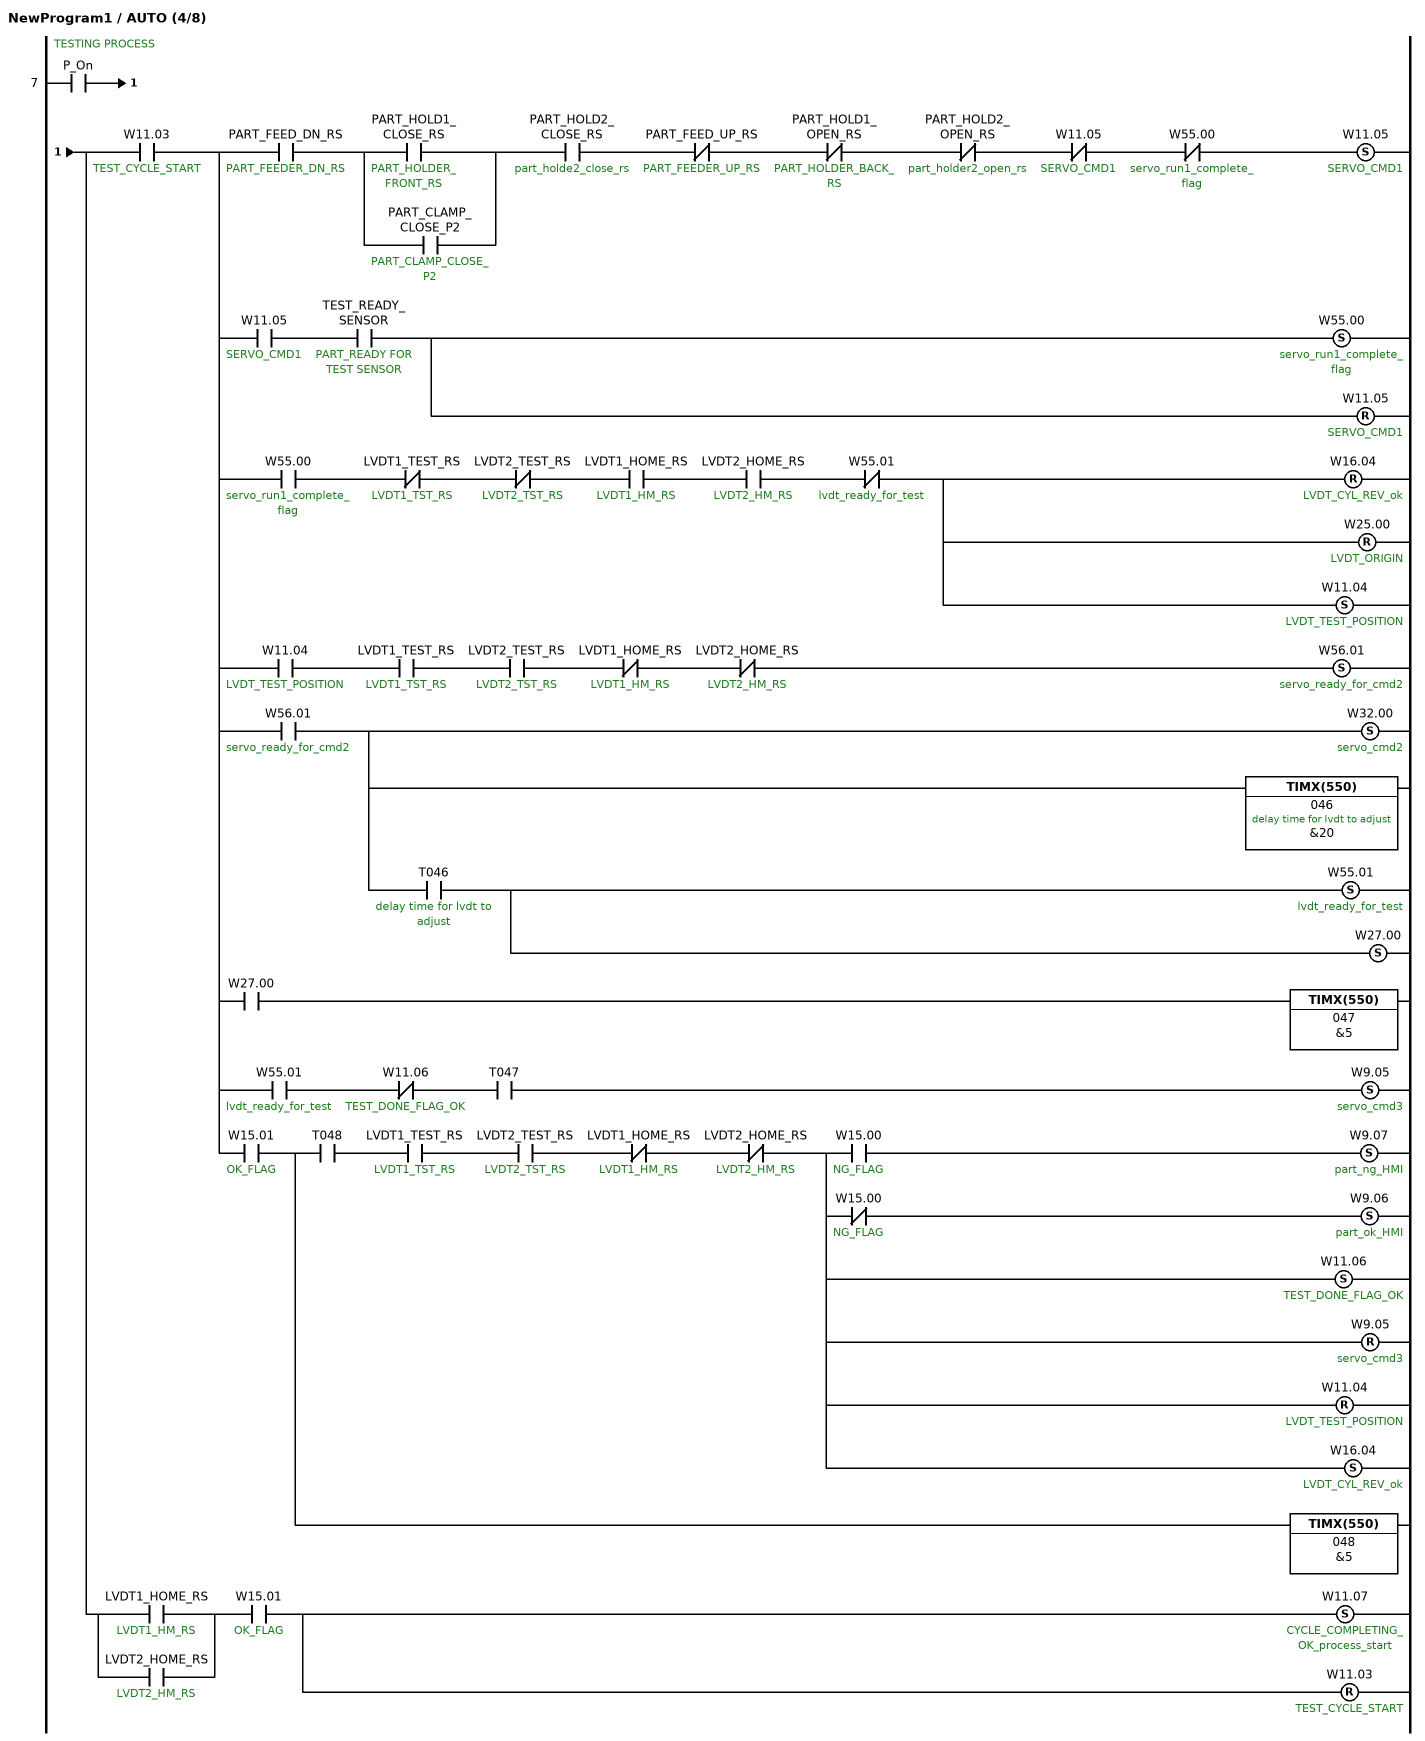
; rung 7: TESTING PROCESS
LD P_On
OUT TR0
AND W11.03  ; TEST_CYCLE_START
OUT TR1
AND PART_FEED_DN_RS  ; PART_FEEDER_DN_RS
LD PART_HOLD1_CLOSE_RS  ; PART_HOLDER_FRONT_RS
OR PART_CLAMP_CLOSE_P2  ; PART_CLAMP_CLOSE_P2
ANDLD
AND PART_HOLD2_CLOSE_RS  ; part_holde2_close_rs
ANDNOT PART_FEED_UP_RS  ; PART_FEEDER_UP_RS
ANDNOT PART_HOLD1_OPEN_RS  ; PART_HOLDER_BACK_RS
ANDNOT PART_HOLD2_OPEN_RS  ; part_holder2_open_rs
ANDNOT W11.05  ; SERVO_CMD1
ANDNOT W55.00  ; servo_run1_complete_flag
SET W11.05  ; SERVO_CMD1
LD TR1
AND W11.05  ; SERVO_CMD1
AND TEST_READY_SENSOR  ; PART_READY FOR TEST SENSOR
SET W55.00  ; servo_run1_complete_flag
RSET W11.05  ; SERVO_CMD1
LD TR1
AND W55.00  ; servo_run1_complete_flag
ANDNOT LVDT1_TEST_RS  ; LVDT1_TST_RS
ANDNOT LVDT2_TEST_RS  ; LVDT2_TST_RS
AND LVDT1_HOME_RS  ; LVDT1_HM_RS
AND LVDT2_HOME_RS  ; LVDT2_HM_RS
ANDNOT W55.01  ; lvdt_ready_for_test
RSET W16.04  ; LVDT_CYL_REV_ok
RSET W25.00  ; LVDT_ORIGIN
SET W11.04  ; LVDT_TEST_POSITION
LD TR1
AND W11.04  ; LVDT_TEST_POSITION
AND LVDT1_TEST_RS  ; LVDT1_TST_RS
AND LVDT2_TEST_RS  ; LVDT2_TST_RS
ANDNOT LVDT1_HOME_RS  ; LVDT1_HM_RS
ANDNOT LVDT2_HOME_RS  ; LVDT2_HM_RS
SET W56.01  ; servo_ready_for_cmd2
LD TR1
AND W56.01  ; servo_ready_for_cmd2
SET W32.00  ; servo_cmd2
TIMX(550) 046 &20  ; delay time for lvdt to adjust
AND T046  ; delay time for lvdt to adjust
SET W55.01  ; lvdt_ready_for_test
SET W27.00
LD TR1
AND W27.00
TIMX(550) 047 &5
LD TR1
AND W55.01  ; lvdt_ready_for_test
ANDNOT W11.06  ; TEST_DONE_FLAG_OK
AND T047
SET W9.05  ; servo_cmd3
LD TR1
AND W15.01  ; OK_FLAG
OUT TR1
AND T048
AND LVDT1_TEST_RS  ; LVDT1_TST_RS
AND LVDT2_TEST_RS  ; LVDT2_TST_RS
ANDNOT LVDT1_HOME_RS  ; LVDT1_HM_RS
ANDNOT LVDT2_HOME_RS  ; LVDT2_HM_RS
OUT TR2
AND W15.00  ; NG_FLAG
SET W9.07  ; part_ng_HMI
LD TR2
ANDNOT W15.00  ; NG_FLAG
SET W9.06  ; part_ok_HMI
LD TR2
SET W11.06  ; TEST_DONE_FLAG_OK
RSET W9.05  ; servo_cmd3
RSET W11.04  ; LVDT_TEST_POSITION
SET W16.04  ; LVDT_CYL_REV_ok
LD TR1
TIMX(550) 048 &5
LD TR0
LD LVDT1_HOME_RS  ; LVDT1_HM_RS
OR LVDT2_HOME_RS  ; LVDT2_HM_RS
ANDLD
AND W15.01  ; OK_FLAG
SET W11.07  ; CYCLE_COMPLETING_OK_process_start
RSET W11.03  ; TEST_CYCLE_START

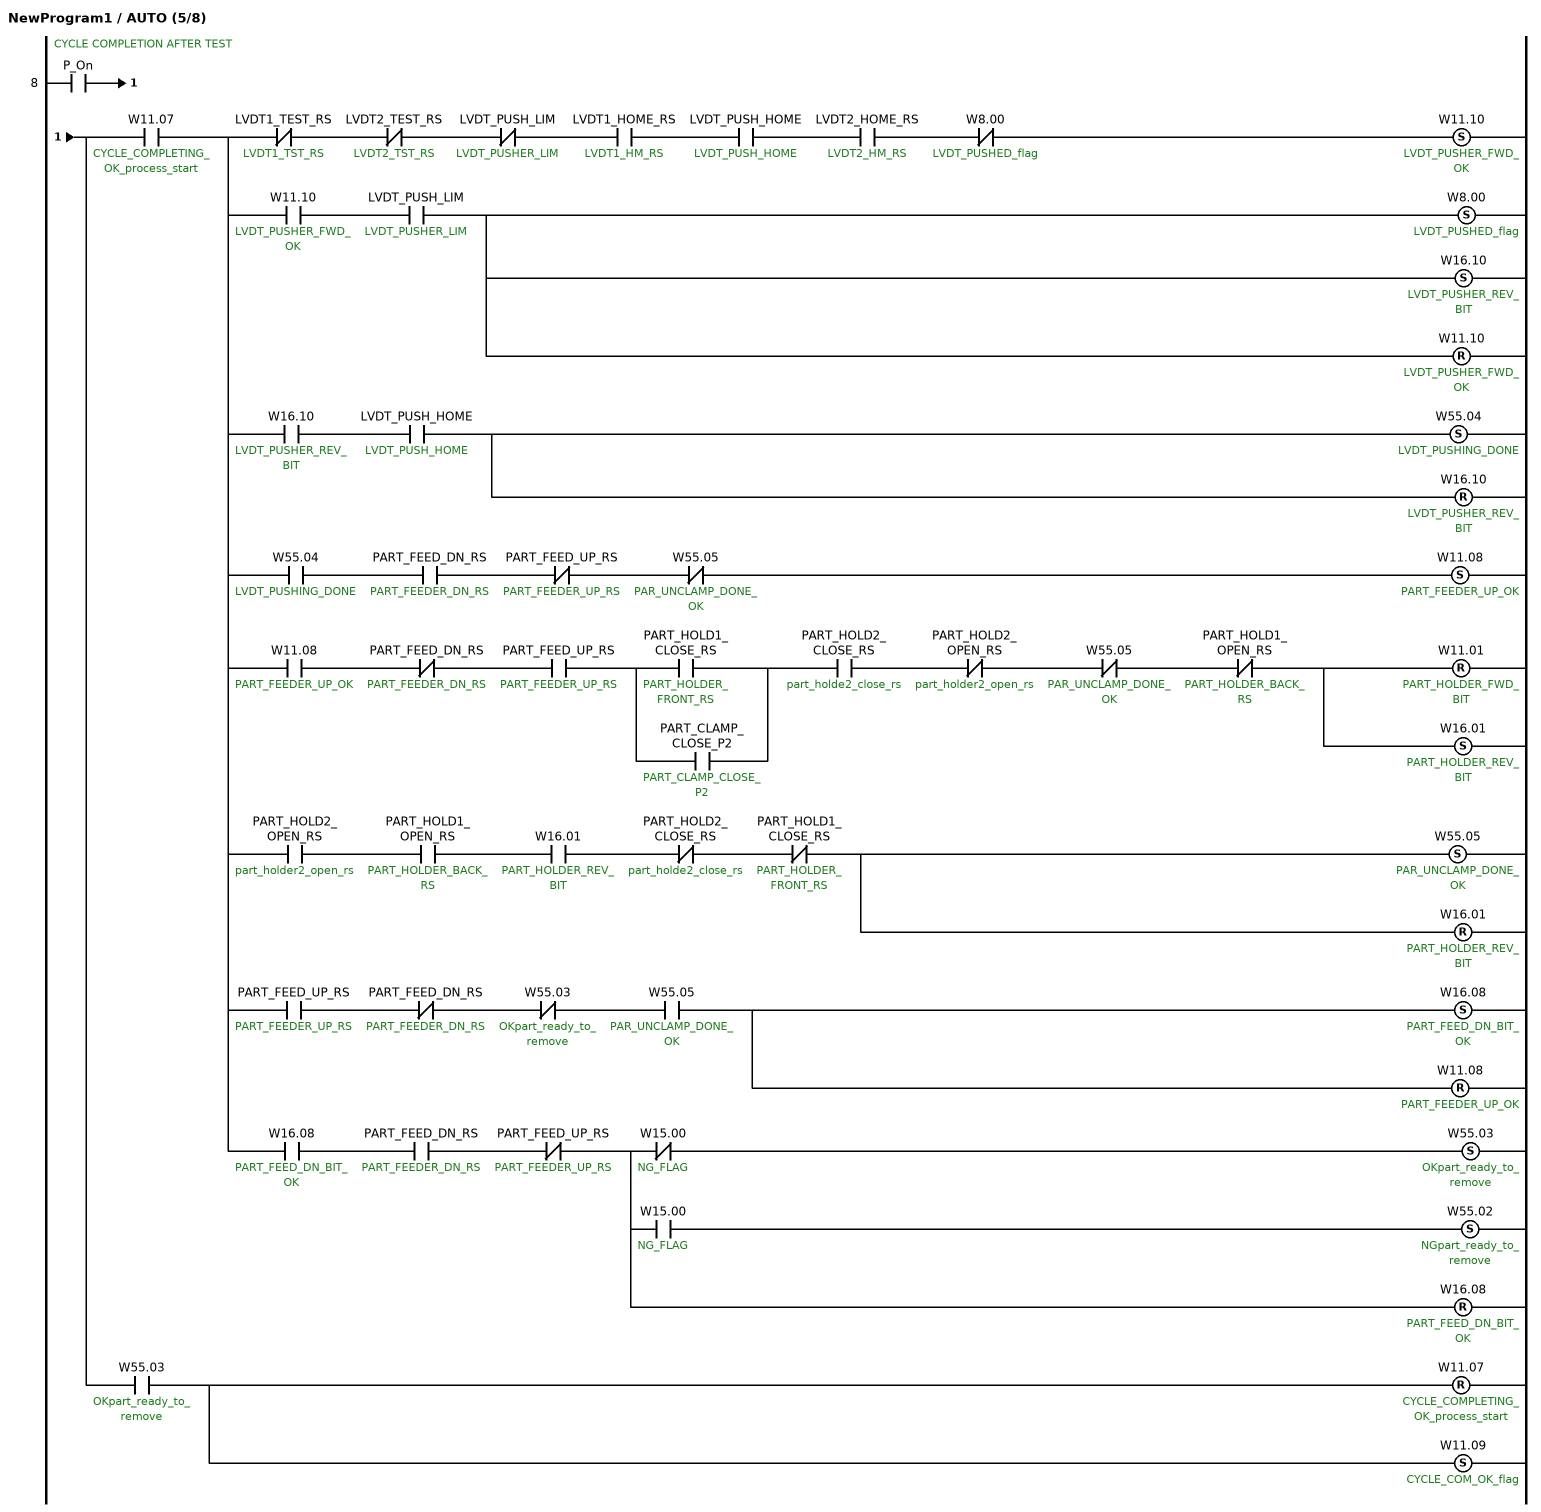
; rung 8: CYCLE COMPLETION AFTER TEST
LD P_On
OUT TR0
AND W11.07  ; CYCLE_COMPLETING_OK_process_start
OUT TR1
ANDNOT LVDT1_TEST_RS  ; LVDT1_TST_RS
ANDNOT LVDT2_TEST_RS  ; LVDT2_TST_RS
ANDNOT LVDT_PUSH_LIM  ; LVDT_PUSHER_LIM
AND LVDT1_HOME_RS  ; LVDT1_HM_RS
AND LVDT_PUSH_HOME  ; LVDT_PUSH_HOME
AND LVDT2_HOME_RS  ; LVDT2_HM_RS
ANDNOT W8.00  ; LVDT_PUSHED_flag
SET W11.10  ; LVDT_PUSHER_FWD_OK
LD TR1
AND W11.10  ; LVDT_PUSHER_FWD_OK
AND LVDT_PUSH_LIM  ; LVDT_PUSHER_LIM
SET W8.00  ; LVDT_PUSHED_flag
SET W16.10  ; LVDT_PUSHER_REV_BIT
RSET W11.10  ; LVDT_PUSHER_FWD_OK
LD TR1
AND W16.10  ; LVDT_PUSHER_REV_BIT
AND LVDT_PUSH_HOME  ; LVDT_PUSH_HOME
SET W55.04  ; LVDT_PUSHING_DONE
RSET W16.10  ; LVDT_PUSHER_REV_BIT
LD TR1
AND W55.04  ; LVDT_PUSHING_DONE
AND PART_FEED_DN_RS  ; PART_FEEDER_DN_RS
ANDNOT PART_FEED_UP_RS  ; PART_FEEDER_UP_RS
ANDNOT W55.05  ; PAR_UNCLAMP_DONE_OK
SET W11.08  ; PART_FEEDER_UP_OK
LD TR1
AND W11.08  ; PART_FEEDER_UP_OK
ANDNOT PART_FEED_DN_RS  ; PART_FEEDER_DN_RS
AND PART_FEED_UP_RS  ; PART_FEEDER_UP_RS
LD PART_HOLD1_CLOSE_RS  ; PART_HOLDER_FRONT_RS
OR PART_CLAMP_CLOSE_P2  ; PART_CLAMP_CLOSE_P2
ANDLD
AND PART_HOLD2_CLOSE_RS  ; part_holde2_close_rs
ANDNOT PART_HOLD2_OPEN_RS  ; part_holder2_open_rs
ANDNOT W55.05  ; PAR_UNCLAMP_DONE_OK
ANDNOT PART_HOLD1_OPEN_RS  ; PART_HOLDER_BACK_RS
RSET W11.01  ; PART_HOLDER_FWD_BIT
SET W16.01  ; PART_HOLDER_REV_BIT
LD TR1
AND PART_HOLD2_OPEN_RS  ; part_holder2_open_rs
AND PART_HOLD1_OPEN_RS  ; PART_HOLDER_BACK_RS
AND W16.01  ; PART_HOLDER_REV_BIT
ANDNOT PART_HOLD2_CLOSE_RS  ; part_holde2_close_rs
ANDNOT PART_HOLD1_CLOSE_RS  ; PART_HOLDER_FRONT_RS
SET W55.05  ; PAR_UNCLAMP_DONE_OK
RSET W16.01  ; PART_HOLDER_REV_BIT
LD TR1
AND PART_FEED_UP_RS  ; PART_FEEDER_UP_RS
ANDNOT PART_FEED_DN_RS  ; PART_FEEDER_DN_RS
ANDNOT W55.03  ; OKpart_ready_to_remove
AND W55.05  ; PAR_UNCLAMP_DONE_OK
SET W16.08  ; PART_FEED_DN_BIT_OK
RSET W11.08  ; PART_FEEDER_UP_OK
LD TR1
AND W16.08  ; PART_FEED_DN_BIT_OK
AND PART_FEED_DN_RS  ; PART_FEEDER_DN_RS
ANDNOT PART_FEED_UP_RS  ; PART_FEEDER_UP_RS
OUT TR1
ANDNOT W15.00  ; NG_FLAG
SET W55.03  ; OKpart_ready_to_remove
LD TR1
AND W15.00  ; NG_FLAG
SET W55.02  ; NGpart_ready_to_remove
LD TR1
RSET W16.08  ; PART_FEED_DN_BIT_OK
LD TR0
AND W55.03  ; OKpart_ready_to_remove
RSET W11.07  ; CYCLE_COMPLETING_OK_process_start
SET W11.09  ; CYCLE_COM_OK_flag

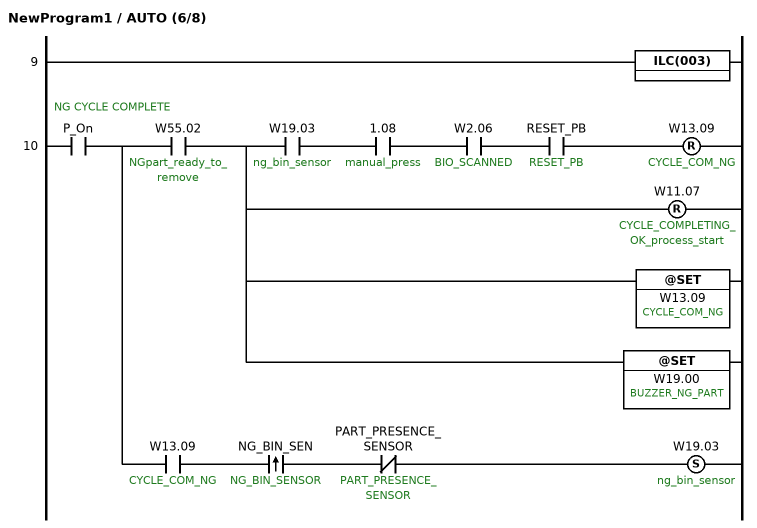
; rung 9
ILC(003)
; rung 10: NG CYCLE COMPLETE
LD P_On
OUT TR0
AND W55.02  ; NGpart_ready_to_remove
OUT TR1
AND W19.03  ; ng_bin_sensor
AND 1.08  ; manual_press
AND W2.06  ; BIO_SCANNED
AND RESET_PB  ; RESET_PB
RSET W13.09  ; CYCLE_COM_NG
LD TR1
RSET W11.07  ; CYCLE_COMPLETING_OK_process_start
@SET W13.09  ; CYCLE_COM_NG
@SET W19.00  ; BUZZER_NG_PART
LD TR0
AND W13.09  ; CYCLE_COM_NG
@AND NG_BIN_SEN  ; NG_BIN_SENSOR
ANDNOT PART_PRESENCE_SENSOR  ; PART_PRESENCE_SENSOR
SET W19.03  ; ng_bin_sensor

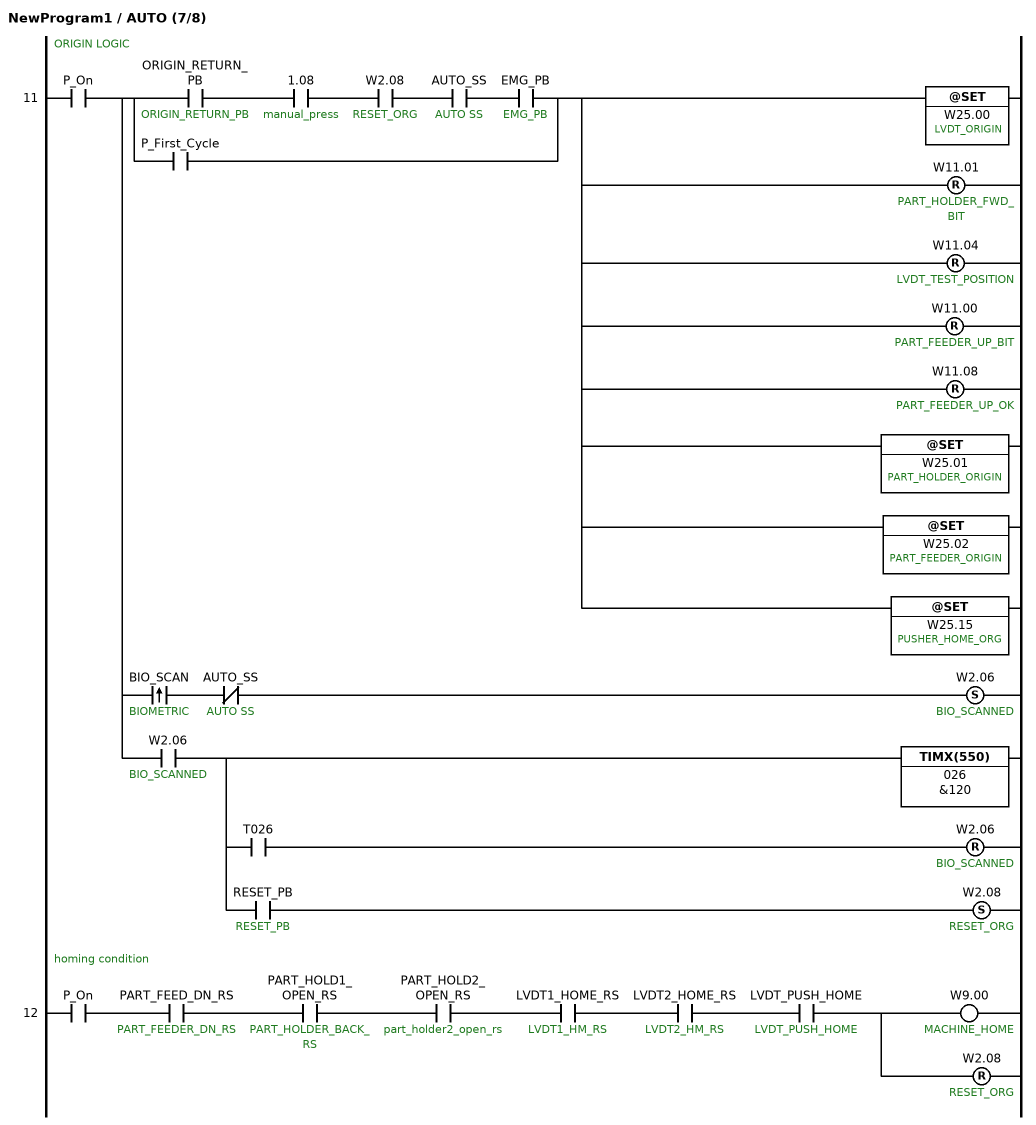
; rung 11: ORIGIN LOGIC
LD P_On
OUT TR0
LD ORIGIN_RETURN_PB  ; ORIGIN_RETURN_PB
AND 1.08  ; manual_press
AND W2.08  ; RESET_ORG
AND AUTO_SS  ; AUTO SS
AND EMG_PB  ; EMG_PB
OR P_First_Cycle
ANDLD
@SET W25.00  ; LVDT_ORIGIN
RSET W11.01  ; PART_HOLDER_FWD_BIT
RSET W11.04  ; LVDT_TEST_POSITION
RSET W11.00  ; PART_FEEDER_UP_BIT
RSET W11.08  ; PART_FEEDER_UP_OK
@SET W25.01  ; PART_HOLDER_ORIGIN
@SET W25.02  ; PART_FEEDER_ORIGIN
@SET W25.15  ; PUSHER_HOME_ORG
LD TR0
@AND BIO_SCAN  ; BIOMETRIC
ANDNOT AUTO_SS  ; AUTO SS
SET W2.06  ; BIO_SCANNED
LD TR0
AND W2.06  ; BIO_SCANNED
OUT TR0
TIMX(550) 026 &120
AND T026
RSET W2.06  ; BIO_SCANNED
LD TR0
AND RESET_PB  ; RESET_PB
SET W2.08  ; RESET_ORG
; rung 12: homing condition
LD P_On
AND PART_FEED_DN_RS  ; PART_FEEDER_DN_RS
AND PART_HOLD1_OPEN_RS  ; PART_HOLDER_BACK_RS
AND PART_HOLD2_OPEN_RS  ; part_holder2_open_rs
AND LVDT1_HOME_RS  ; LVDT1_HM_RS
AND LVDT2_HOME_RS  ; LVDT2_HM_RS
AND LVDT_PUSH_HOME  ; LVDT_PUSH_HOME
OUT W9.00  ; MACHINE_HOME
RSET W2.08  ; RESET_ORG

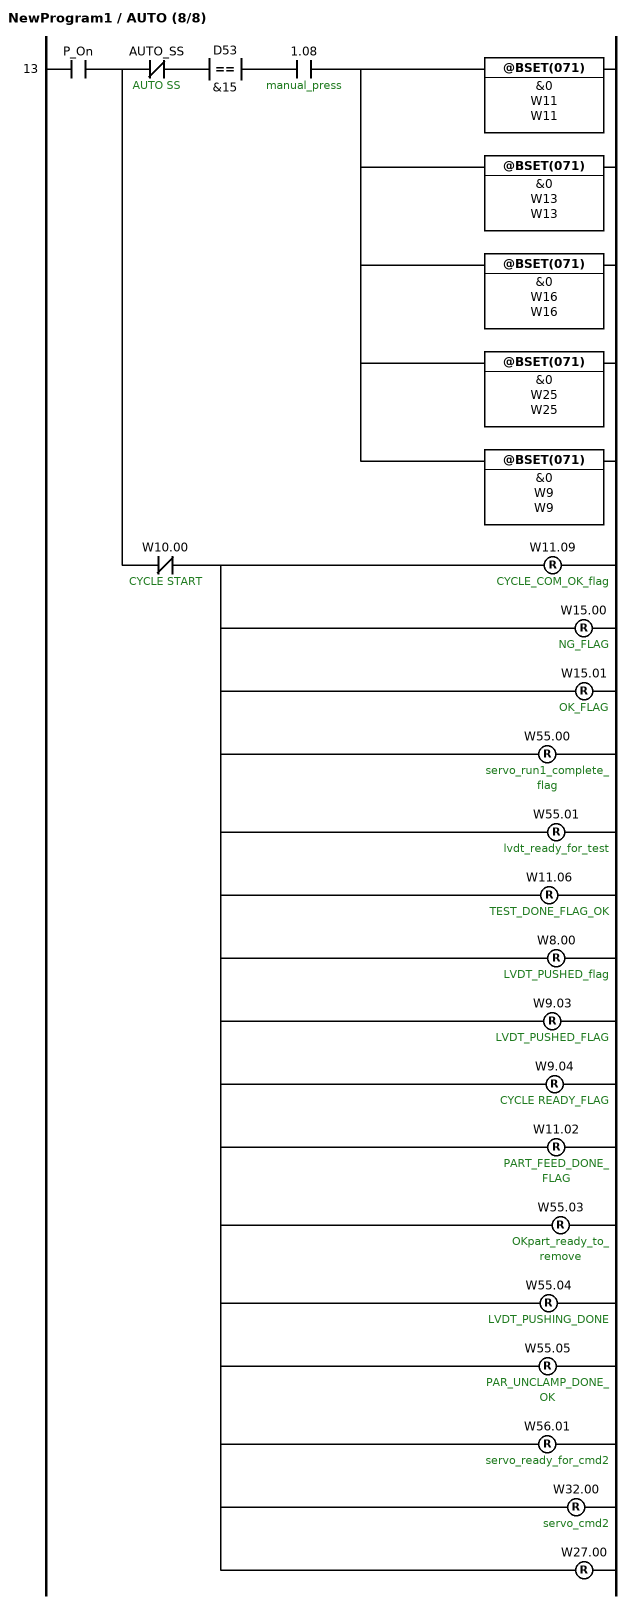
; rung 13
LD P_On
OUT TR0
ANDNOT AUTO_SS  ; AUTO SS
AND=(300) D53 &15
AND 1.08  ; manual_press
@BSET(071) &0 W11 W11
@BSET(071) &0 W13 W13
@BSET(071) &0 W16 W16
@BSET(071) &0 W25 W25
@BSET(071) &0 W9 W9
LD TR0
ANDNOT W10.00  ; CYCLE START
RSET W11.09  ; CYCLE_COM_OK_flag
RSET W15.00  ; NG_FLAG
RSET W15.01  ; OK_FLAG
RSET W55.00  ; servo_run1_complete_flag
RSET W55.01  ; lvdt_ready_for_test
RSET W11.06  ; TEST_DONE_FLAG_OK
RSET W8.00  ; LVDT_PUSHED_flag
RSET W9.03  ; LVDT_PUSHED_FLAG
RSET W9.04  ; CYCLE READY_FLAG
RSET W11.02  ; PART_FEED_DONE_FLAG
RSET W55.03  ; OKpart_ready_to_remove
RSET W55.04  ; LVDT_PUSHING_DONE
RSET W55.05  ; PAR_UNCLAMP_DONE_OK
RSET W56.01  ; servo_ready_for_cmd2
RSET W32.00  ; servo_cmd2
RSET W27.00

### Section LVDT_CAL

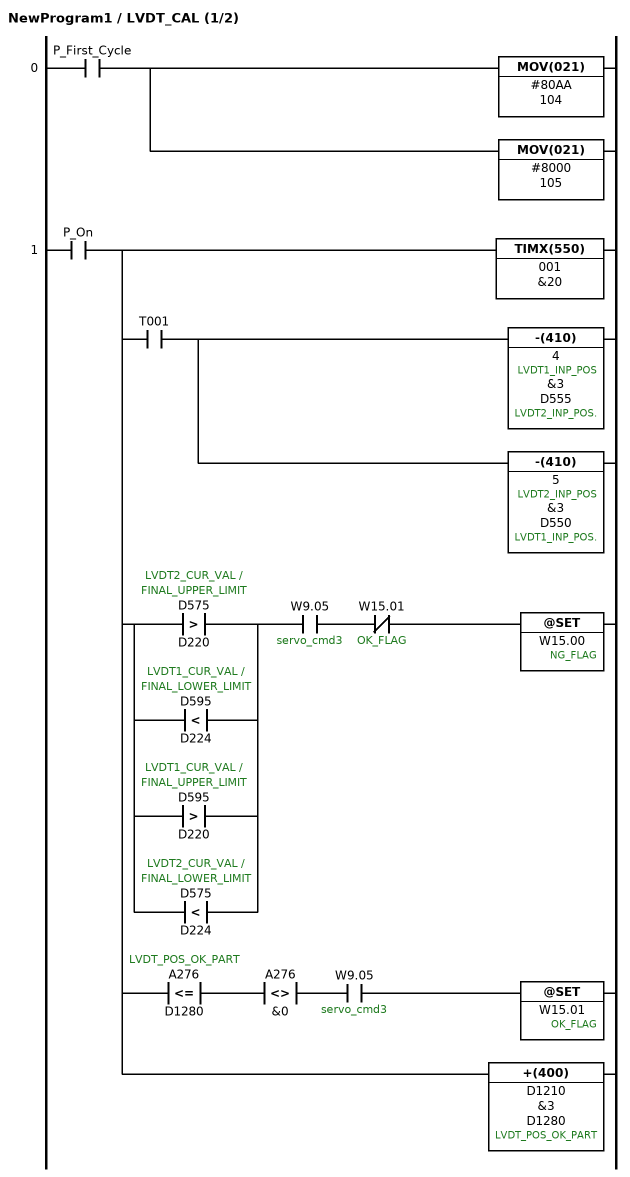
; rung 0
LD P_First_Cycle
MOV(021) #80AA 104
MOV(021) #8000 105
; rung 1
LD P_On
OUT TR0
TIMX(550) 001 &20
AND T001
-(410) 4 &3 D555  ; LVDT1_INP_POS, LVDT2_INP_POS.
-(410) 5 &3 D550  ; LVDT2_INP_POS, LVDT1_INP_POS.
LD TR0
LD>F(333) D575 D220  ; LVDT2_CUR_VAL, FINAL_UPPER_LIMIT
OR<F(331) D595 D224  ; LVDT1_CUR_VAL, FINAL_LOWER_LIMIT
OR>F(333) D595 D220  ; LVDT1_CUR_VAL, FINAL_UPPER_LIMIT
OR<F(331) D575 D224  ; LVDT2_CUR_VAL, FINAL_LOWER_LIMIT
ANDLD
AND W9.05  ; servo_cmd3
ANDNOT W15.01  ; OK_FLAG
@SET W15.00  ; NG_FLAG
LD TR0
AND<=(315) A276 D1280  ; LVDT_POS_OK_PART
AND<>(305) A276 &0
AND W9.05  ; servo_cmd3
@SET W15.01  ; OK_FLAG
LD TR0
+(400) D1210 &3 D1280  ; LVDT_POS_OK_PART

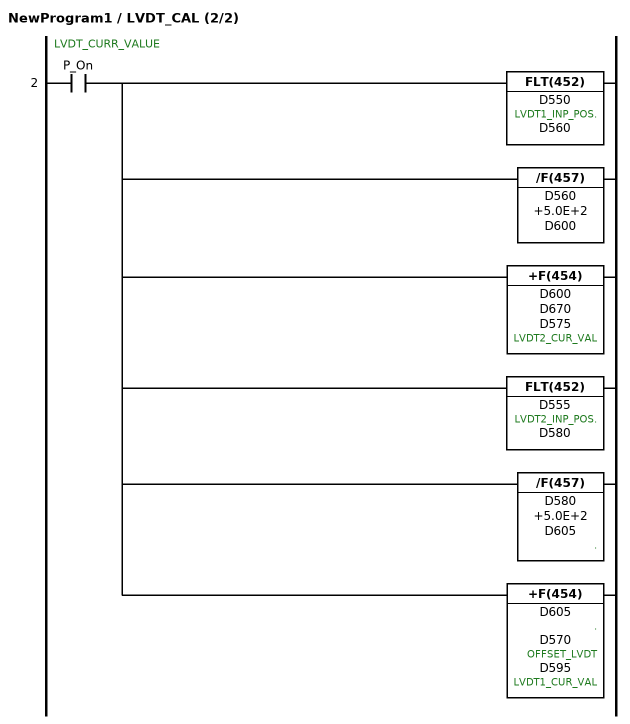
; rung 2: LVDT_CURR_VALUE
LD P_On
FLT(452) D550 D560  ; LVDT1_INP_POS.
/F(457) D560 +5.0E+2 D600
+F(454) D600 D670 D575  ; LVDT2_CUR_VAL
FLT(452) D555 D580  ; LVDT2_INP_POS.
/F(457) D580 +5.0E+2 D605  ; .
+F(454) D605 D570 D595  ; ., OFFSET_LVDT, LVDT1_CUR_VAL

### Section MODEL_SELECTION

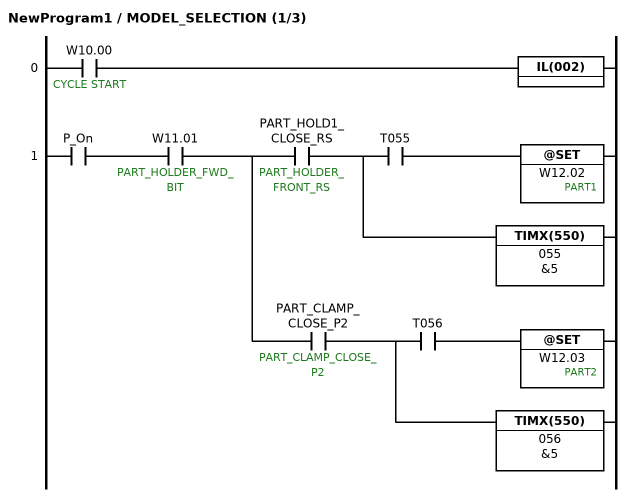
; rung 0
LD W10.00  ; CYCLE START
IL(002)
; rung 1
LD P_On
AND W11.01  ; PART_HOLDER_FWD_BIT
OUT TR0
AND PART_HOLD1_CLOSE_RS  ; PART_HOLDER_FRONT_RS
OUT TR1
AND T055
@SET W12.02  ; PART1
LD TR1
TIMX(550) 055 &5
LD TR0
AND PART_CLAMP_CLOSE_P2  ; PART_CLAMP_CLOSE_P2
OUT TR0
AND T056
@SET W12.03  ; PART2
LD TR0
TIMX(550) 056 &5

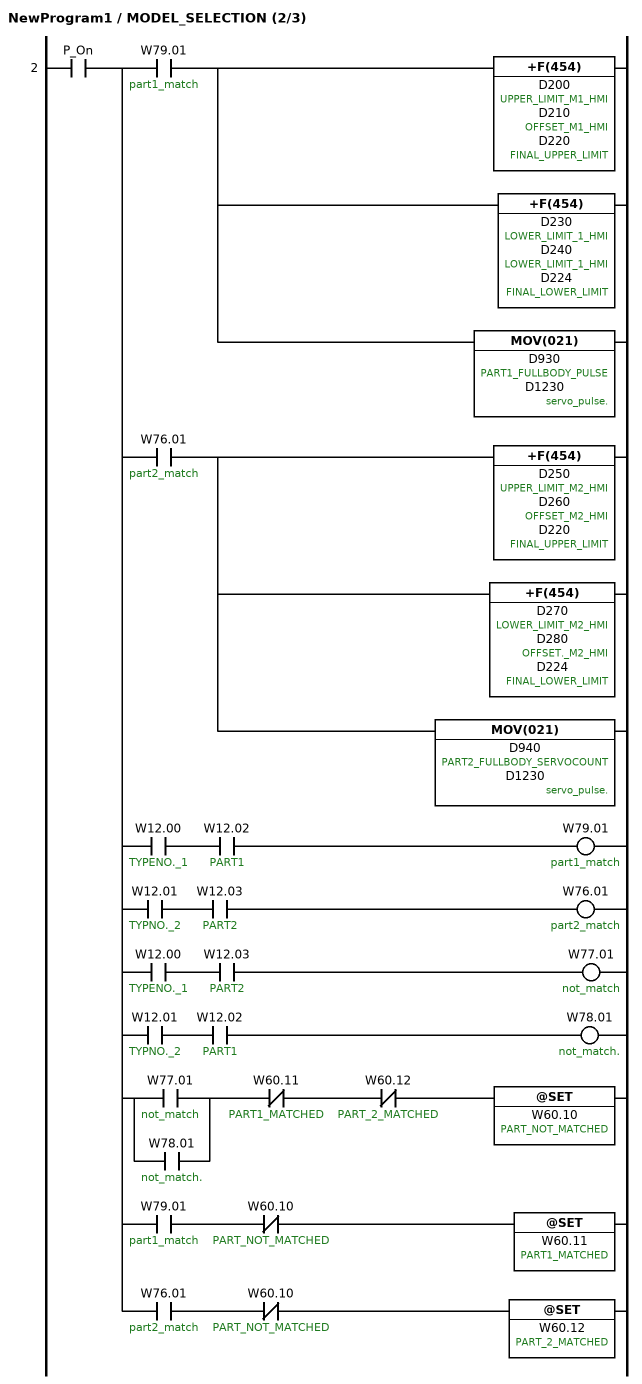
; rung 2
LD P_On
OUT TR0
AND W79.01  ; part1_match
+F(454) D200 D210 D220  ; UPPER_LIMIT_M1_HMI, OFFSET_M1_HMI, FINAL_UPPER_LIMIT
+F(454) D230 D240 D224  ; LOWER_LIMIT_1_HMI, FINAL_LOWER_LIMIT
MOV(021) D930 D1230  ; PART1_FULLBODY_PULSE, servo_pulse.
LD TR0
AND W76.01  ; part2_match
+F(454) D250 D260 D220  ; UPPER_LIMIT_M2_HMI, OFFSET_M2_HMI, FINAL_UPPER_LIMIT
+F(454) D270 D280 D224  ; LOWER_LIMIT_M2_HMI, OFFSET._M2_HMI, FINAL_LOWER_LIMIT
MOV(021) D940 D1230  ; PART2_FULLBODY_SERVOCOUNT, servo_pulse.
LD TR0
AND W12.00  ; TYPENO._1
AND W12.02  ; PART1
OUT W79.01  ; part1_match
LD TR0
AND W12.01  ; TYPNO._2
AND W12.03  ; PART2
OUT W76.01  ; part2_match
LD TR0
AND W12.00  ; TYPENO._1
AND W12.03  ; PART2
OUT W77.01  ; not_match
LD TR0
AND W12.01  ; TYPNO._2
AND W12.02  ; PART1
OUT W78.01  ; not_match.
LD TR0
LD W77.01  ; not_match
OR W78.01  ; not_match.
ANDLD
ANDNOT W60.11  ; PART1_MATCHED
ANDNOT W60.12  ; PART_2_MATCHED
@SET W60.10  ; PART_NOT_MATCHED
LD TR0
AND W79.01  ; part1_match
ANDNOT W60.10  ; PART_NOT_MATCHED
@SET W60.11  ; PART1_MATCHED
LD TR0
AND W76.01  ; part2_match
ANDNOT W60.10  ; PART_NOT_MATCHED
@SET W60.12  ; PART_2_MATCHED

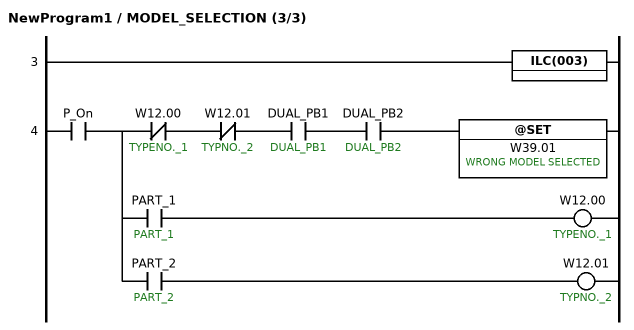
; rung 3
ILC(003)
; rung 4
LD P_On
OUT TR0
ANDNOT W12.00  ; TYPENO._1
ANDNOT W12.01  ; TYPNO._2
AND DUAL_PB1  ; DUAL_PB1
AND DUAL_PB2  ; DUAL_PB2
@SET W39.01  ; WRONG MODEL SELECTED
LD TR0
AND PART_1  ; PART_1
OUT W12.00  ; TYPENO._1
LD TR0
AND PART_2  ; PART_2
OUT W12.01  ; TYPNO._2

### Section ALARMS

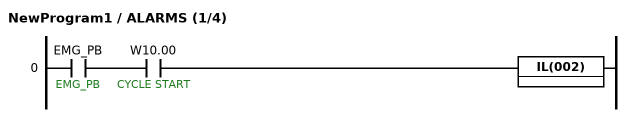
; rung 0
LD EMG_PB  ; EMG_PB
AND W10.00  ; CYCLE START
IL(002)

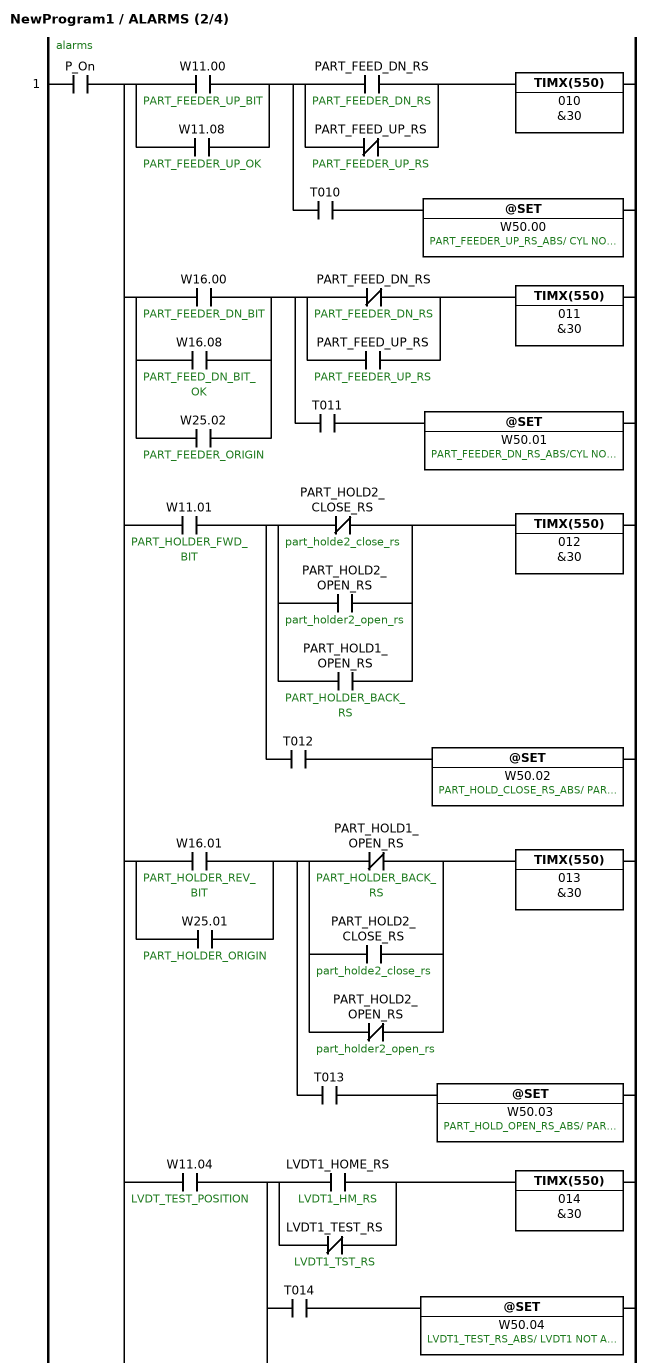

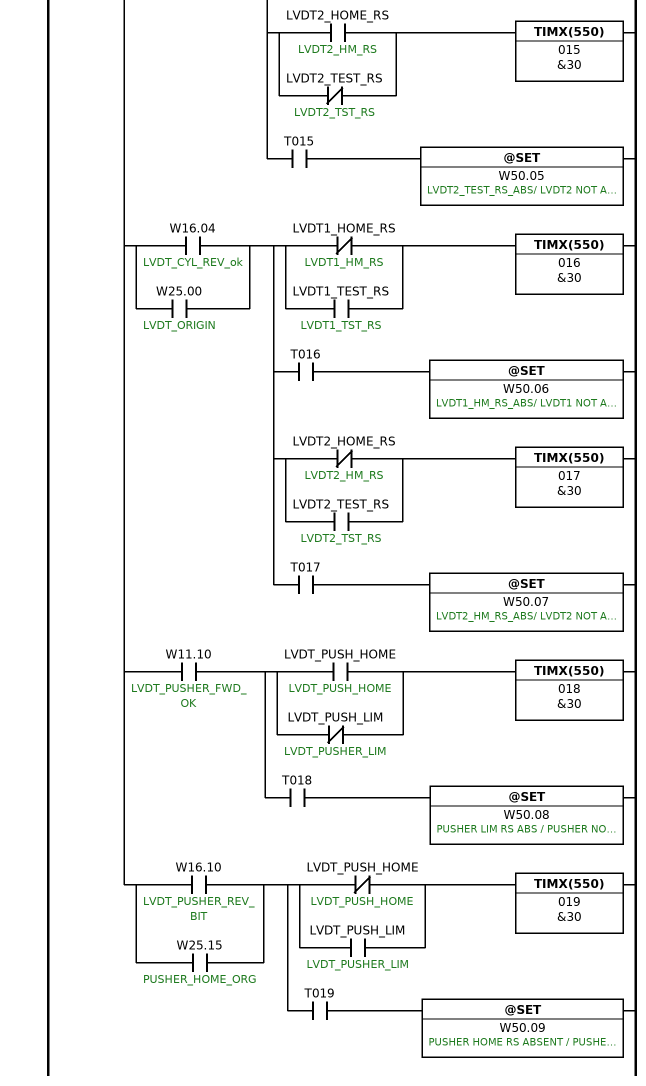
; rung 1: alarms
LD P_On
OUT TR0
LD W11.00  ; PART_FEEDER_UP_BIT
OR W11.08  ; PART_FEEDER_UP_OK
ANDLD
OUT TR1
LD PART_FEED_DN_RS  ; PART_FEEDER_DN_RS
ORNOT PART_FEED_UP_RS  ; PART_FEEDER_UP_RS
ANDLD
TIMX(550) 010 &30
LD TR1
AND T010
@SET W50.00  ; PART_FEEDER_UP_RS_ABS/ CYL NOT UP
LD TR0
LD W16.00  ; PART_FEEDER_DN_BIT
OR W16.08  ; PART_FEED_DN_BIT_OK
OR W25.02  ; PART_FEEDER_ORIGIN
ANDLD
OUT TR1
LDNOT PART_FEED_DN_RS  ; PART_FEEDER_DN_RS
OR PART_FEED_UP_RS  ; PART_FEEDER_UP_RS
ANDLD
TIMX(550) 011 &30
LD TR1
AND T011
@SET W50.01  ; PART_FEEDER_DN_RS_ABS/CYL NOT DN
LD TR0
AND W11.01  ; PART_HOLDER_FWD_BIT
OUT TR1
LDNOT PART_HOLD2_CLOSE_RS  ; part_holde2_close_rs
OR PART_HOLD2_OPEN_RS  ; part_holder2_open_rs
OR PART_HOLD1_OPEN_RS  ; PART_HOLDER_BACK_RS
ANDLD
TIMX(550) 012 &30
LD TR1
AND T012
@SET W50.02  ; PART_HOLD_CLOSE_RS_ABS/ PART NOT HOLD
LD TR0
LD W16.01  ; PART_HOLDER_REV_BIT
OR W25.01  ; PART_HOLDER_ORIGIN
ANDLD
OUT TR1
LDNOT PART_HOLD1_OPEN_RS  ; PART_HOLDER_BACK_RS
OR PART_HOLD2_CLOSE_RS  ; part_holde2_close_rs
ORNOT PART_HOLD2_OPEN_RS  ; part_holder2_open_rs
ANDLD
TIMX(550) 013 &30
LD TR1
AND T013
@SET W50.03  ; PART_HOLD_OPEN_RS_ABS/ PART NOT RELEASED
LD TR0
AND W11.04  ; LVDT_TEST_POSITION
OUT TR1
LD LVDT1_HOME_RS  ; LVDT1_HM_RS
ORNOT LVDT1_TEST_RS  ; LVDT1_TST_RS
ANDLD
TIMX(550) 014 &30
LD TR1
AND T014
@SET W50.04  ; LVDT1_TEST_RS_ABS/ LVDT1 NOT AT TEST POS
LD TR1
LD LVDT2_HOME_RS  ; LVDT2_HM_RS
ORNOT LVDT2_TEST_RS  ; LVDT2_TST_RS
ANDLD
TIMX(550) 015 &30
LD TR1
AND T015
@SET W50.05  ; LVDT2_TEST_RS_ABS/ LVDT2 NOT AT TEST POS
LD TR0
LD W16.04  ; LVDT_CYL_REV_ok
OR W25.00  ; LVDT_ORIGIN
ANDLD
OUT TR1
LDNOT LVDT1_HOME_RS  ; LVDT1_HM_RS
OR LVDT1_TEST_RS  ; LVDT1_TST_RS
ANDLD
TIMX(550) 016 &30
LD TR1
AND T016
@SET W50.06  ; LVDT1_HM_RS_ABS/ LVDT1 NOT AT HOME POS
LD TR1
LDNOT LVDT2_HOME_RS  ; LVDT2_HM_RS
OR LVDT2_TEST_RS  ; LVDT2_TST_RS
ANDLD
TIMX(550) 017 &30
LD TR1
AND T017
@SET W50.07  ; LVDT2_HM_RS_ABS/ LVDT2 NOT AT HOME POS
LD TR0
AND W11.10  ; LVDT_PUSHER_FWD_OK
OUT TR1
LD LVDT_PUSH_HOME  ; LVDT_PUSH_HOME
ORNOT LVDT_PUSH_LIM  ; LVDT_PUSHER_LIM
ANDLD
TIMX(550) 018 &30
LD TR1
AND T018
@SET W50.08  ; PUSHER LIM RS ABS / PUSHER NOT MOVING FWD
LD TR0
LD W16.10  ; LVDT_PUSHER_REV_BIT
OR W25.15  ; PUSHER_HOME_ORG
ANDLD
OUT TR0
LDNOT LVDT_PUSH_HOME  ; LVDT_PUSH_HOME
OR LVDT_PUSH_LIM  ; LVDT_PUSHER_LIM
ANDLD
TIMX(550) 019 &30
LD TR0
AND T019
@SET W50.09  ; PUSHER HOME RS ABSENT / PUSHER NOT MOVING REV

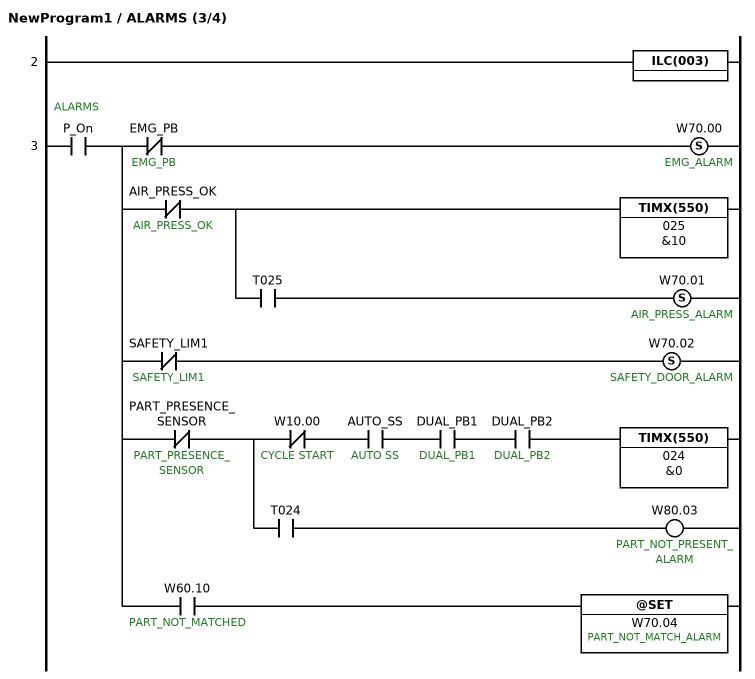
; rung 2
ILC(003)
; rung 3: ALARMS
LD P_On
OUT TR0
ANDNOT EMG_PB  ; EMG_PB
SET W70.00  ; EMG_ALARM
LD TR0
ANDNOT AIR_PRESS_OK  ; AIR_PRESS_OK
TIMX(550) 025 &10
AND T025
SET W70.01  ; AIR_PRESS_ALARM
LD TR0
ANDNOT SAFETY_LIM1  ; SAFETY_LIM1
SET W70.02  ; SAFETY_DOOR_ALARM
LD TR0
ANDNOT PART_PRESENCE_SENSOR  ; PART_PRESENCE_SENSOR
OUT TR1
ANDNOT W10.00  ; CYCLE START
AND AUTO_SS  ; AUTO SS
AND DUAL_PB1  ; DUAL_PB1
AND DUAL_PB2  ; DUAL_PB2
TIMX(550) 024 &0
LD TR1
AND T024
OUT W80.03  ; PART_NOT_PRESENT_ALARM
LD TR0
AND W60.10  ; PART_NOT_MATCHED
@SET W70.04  ; PART_NOT_MATCH_ALARM

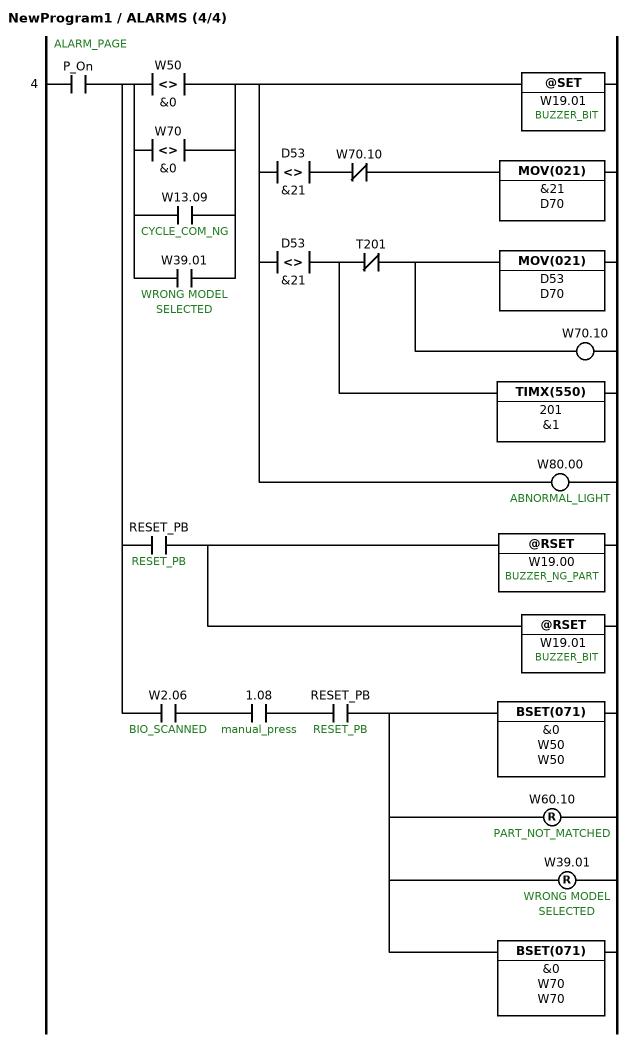
; rung 4: ALARM_PAGE
LD P_On
OUT TR0
LD<>(305) W50 &0
OR<>(305) W70 &0
OR W13.09  ; CYCLE_COM_NG
OR W39.01  ; WRONG MODEL SELECTED
ANDLD
OUT TR1
@SET W19.01  ; BUZZER_BIT
AND<>(305) D53 &21
ANDNOT W70.10
MOV(021) &21 D70
LD TR1
AND<>(305) D53 &21
OUT TR2
ANDNOT T201
MOV(021) D53 D70
OUT W70.10
LD TR2
TIMX(550) 201 &1
LD TR1
OUT W80.00  ; ABNORMAL_LIGHT
LD TR0
AND RESET_PB  ; RESET_PB
@RSET W19.00  ; BUZZER_NG_PART
@RSET W19.01  ; BUZZER_BIT
LD TR0
AND W2.06  ; BIO_SCANNED
AND 1.08  ; manual_press
AND RESET_PB  ; RESET_PB
BSET(071) &0 W50 W50
RSET W60.10  ; PART_NOT_MATCHED
RSET W39.01  ; WRONG MODEL SELECTED
BSET(071) &0 W70 W70

### Section SERVO

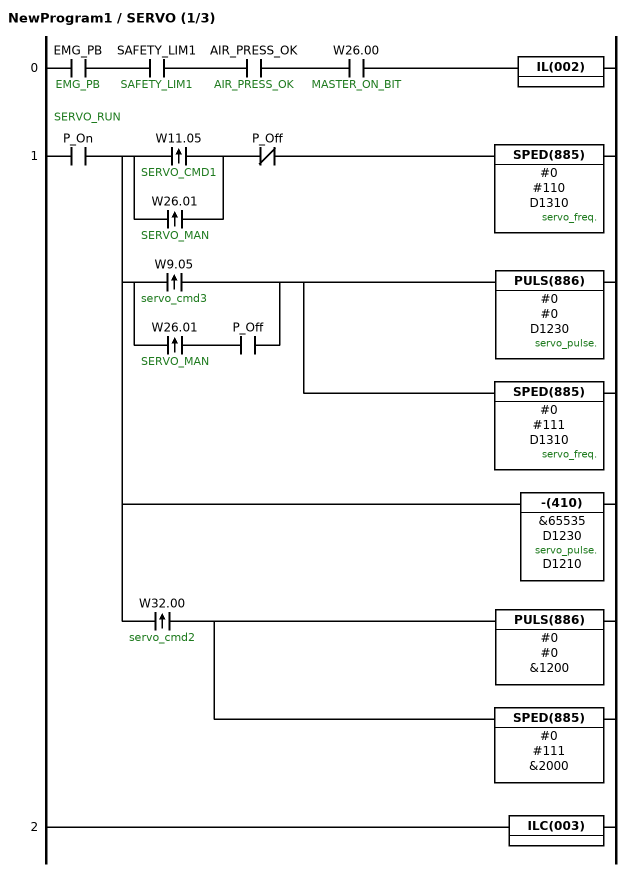
; rung 0
LD EMG_PB  ; EMG_PB
AND SAFETY_LIM1  ; SAFETY_LIM1
AND AIR_PRESS_OK  ; AIR_PRESS_OK
AND W26.00  ; MASTER_ON_BIT
IL(002)
; rung 1: SERVO_RUN
LD P_On
OUT TR0
@LD W11.05  ; SERVO_CMD1
@OR W26.01  ; SERVO_MAN
ANDLD
ANDNOT P_Off
SPED(885) #0 #110 D1310  ; servo_freq.
LD TR0
@LD W9.05  ; servo_cmd3
@LD W26.01  ; SERVO_MAN
AND P_Off
ORLD
ANDLD
PULS(886) #0 #0 D1230  ; servo_pulse.
SPED(885) #0 #111 D1310  ; servo_freq.
LD TR0
-(410) &65535 D1230 D1210  ; servo_pulse.
@AND W32.00  ; servo_cmd2
PULS(886) #0 #0 &1200
SPED(885) #0 #111 &2000
; rung 2
ILC(003)

